C03645=1190.847,-75.511,-40.674,179.388,5.625,149.176
C03646=1190.842,-75.240,-40.686,179.390,5.625,149.175
C03647=1190.836,-74.969,-40.698,179.392,5.625,149.174
C03648=1190.830,-74.720,-40.709,179.395,5.625,149.173
C03649=1190.826,-74.470,-40.720,179.397,5.625,149.173
C03650=1190.820,-74.220,-40.730,179.399,5.626,149.172
C03651=1190.815,-73.970,-40.741,179.402,5.626,149.172
C03652=1190.810,-73.721,-40.752,179.404,5.626,149.171
C03653=1190.804,-73.471,-40.763,179.406,5.627,149.170
C03654=1190.799,-73.222,-40.774,179.409,5.627,149.170
C03655=1190.794,-72.972,-40.784,179.411,5.627,149.169
C03656=1190.789,-72.722,-40.796,179.413,5.627,149.168
C03657=1190.783,-72.472,-40.806,179.415,5.627,149.168
C03658=1190.779,-72.223,-40.817,179.418,5.628,149.167
C03659=1190.772,-71.973,-40.828,179.420,5.628,149.167
C03660=1190.768,-71.723,-40.839,179.422,5.628,149.166
C03661=1190.763,-71.473,-40.850,179.425,5.628,149.165
C03662=1190.757,-71.224,-40.861,179.428,5.629,149.164
C03663=1190.752,-70.974,-40.871,179.429,5.629,149.164
C03664=1190.746,-70.725,-40.883,179.432,5.629,149.163
C03665=1190.741,-70.474,-40.893,179.435,5.630,149.163
C03666=1190.737,-70.225,-40.905,179.436,5.630,149.162
C03667=1190.731,-69.976,-40.915,179.439,5.630,149.161
C03668=1190.726,-69.725,-40.927,179.441,5.630,149.161
C03669=1190.720,-69.476,-40.938,179.444,5.630,149.160
C03670=1190.715,-69.226,-40.948,179.446,5.631,149.159
C03671=1190.711,-68.976,-40.959,179.448,5.631,149.159
C03672=1190.704,-68.727,-40.970,179.451,5.631,149.158
C03673=1190.700,-68.477,-40.982,179.453,5.632,149.158
C03674=1190.695,-68.227,-40.993,179.455,5.631,149.157
C03675=1190.689,-67.978,-41.003,179.457,5.632,149.156
C03676=1190.684,-67.728,-41.015,179.460,5.632,149.155
C03677=1190.679,-67.478,-41.026,179.462,5.632,149.155
C03678=1190.674,-67.229,-41.036,179.464,5.633,149.154
C03679=1190.668,-66.979,-41.048,179.466,5.632,149.154
C03680=1190.663,-66.729,-41.059,179.469,5.633,149.153
C03681=1190.658,-66.480,-41.070,179.471,5.634,149.152
C03682=1190.653,-66.230,-41.081,179.473,5.633,149.152
C03683=1190.648,-65.979,-41.092,179.476,5.634,149.151
C03684=1190.642,-65.731,-41.103,179.478,5.634,149.151
C03685=1190.638,-65.481,-41.114,179.480,5.634,149.150
C03686=1190.632,-65.230,-41.126,179.483,5.635,149.149
C03687=1190.626,-64.981,-41.137,179.486,5.635,149.148
C03688=1190.622,-64.732,-41.148,179.487,5.635,149.148
C03689=1190.616,-64.482,-41.160,179.490,5.635,149.147
C03690=1190.611,-64.232,-41.170,179.493,5.636,149.147
C03691=1190.606,-63.983,-41.181,179.494,5.636,149.146
C03692=1190.601,-63.733,-41.193,179.497,5.636,149.145
C03693=1190.595,-63.484,-41.204,179.500,5.637,149.145
C03694=1190.590,-63.233,-41.215,179.502,5.636,149.144
C03695=1190.585,-62.984,-41.227,179.504,5.637,149.143
C03696=1190.580,-62.734,-41.238,179.506,5.638,149.143
C03697=1190.574,-62.485,-41.249,179.509,5.637,149.142
C03698=1190.569,-62.235,-41.260,179.511,5.638,149.141
C03699=1190.565,-61.985,-41.271,179.513,5.638,149.141
C03700=1190.559,-61.735,-41.283,179.515,5.638,149.140
C03701=1190.554,-61.486,-41.294,179.518,5.638,149.139
C03702=1190.548,-61.236,-41.306,179.520,5.639,149.139
C03703=1190.543,-60.986,-41.316,179.522,5.639,149.138
C03704=1190.539,-60.736,-41.328,179.525,5.639,149.138
C03705=1190.533,-60.487,-41.339,179.528,5.640,149.137
C03706=1190.528,-60.237,-41.351,179.529,5.640,149.136
C03707=1190.523,-59.987,-41.362,179.532,5.640,149.136
C03708=1190.518,-59.738,-41.374,179.535,5.641,149.135
C03709=1190.512,-59.488,-41.385,179.537,5.640,149.134
C03710=1190.507,-59.238,-41.396,179.539,5.641,149.134
C03711=1190.501,-58.988,-41.408,179.542,5.642,149.133
C03712=1190.497,-58.739,-41.419,179.544,5.641,149.132
C03713=1190.491,-58.490,-41.430,179.546,5.642,149.132
C03714=1190.486,-58.240,-41.442,179.549,5.642,149.131
C03715=1190.481,-57.990,-41.453,179.551,5.642,149.130
C03716=1190.476,-57.740,-41.465,179.553,5.642,149.130
C03717=1190.471,-57.491,-41.476,179.556,5.643,149.129
C03718=1190.465,-57.242,-41.488,179.558,5.643,149.129
C03719=1190.460,-56.991,-41.498,179.560,5.643,149.128
C03720=1190.455,-56.741,-41.510,179.563,5.644,149.127
C03721=1190.450,-56.492,-41.522,179.565,5.645,149.127
C03722=1190.445,-56.242,-41.533,179.567,5.644,149.126
C03723=1190.440,-55.992,-41.545,179.570,5.645,149.125
C03724=1190.434,-55.743,-41.556,179.573,5.645,149.125
C03725=1190.429,-55.493,-41.568,179.574,5.645,149.124
C03726=1190.424,-55.243,-41.579,179.577,5.646,149.123
C03727=1190.419,-54.994,-41.591,179.579,5.646,149.123
C03728=1190.414,-54.744,-41.603,179.581,5.646,149.122
C03729=1190.409,-54.494,-41.614,179.584,5.646,149.122
C03730=1190.403,-54.245,-41.625,179.586,5.647,149.121
C03731=1190.397,-53.995,-41.637,179.588,5.647,149.120
C03732=1190.393,-53.745,-41.649,179.591,5.647,149.119
C03733=1190.387,-53.495,-41.660,179.593,5.648,149.119
C03734=1190.383,-53.246,-41.672,179.596,5.648,149.118
C03735=1190.377,-52.996,-41.684,179.598,5.648,149.118
C03736=1190.373,-52.746,-41.695,179.601,5.648,149.117
C03737=1190.367,-52.498,-41.707,179.603,5.649,149.116
C03738=1190.361,-52.248,-41.719,179.605,5.649,149.116
C03739=1190.357,-51.998,-41.730,179.608,5.649,149.115
C03740=1190.351,-51.748,-41.742,179.610,5.650,149.114
C03741=1190.347,-51.498,-41.754,179.612,5.650,149.114
C03742=1190.341,-51.249,-41.765,179.615,5.650,149.113
C03743=1190.336,-50.999,-41.777,179.617,5.651,149.112
C03744=1190.331,-50.749,-41.789,179.620,5.651,149.112
C03745=1190.325,-50.500,-41.800,179.621,5.651,149.111
C03746=1190.320,-50.250,-41.812,179.624,5.651,149.110
C03747=1190.315,-50.001,-41.824,179.627,5.652,149.110
C03748=1190.310,-49.730,-41.836,179.629,5.652,149.109
C03749=1190.304,-49.460,-41.849,179.632,5.652,149.108
C03750=1190.298,-49.190,-41.862,179.634,5.652,149.108
C03751=1190.293,-48.919,-41.875,179.637,5.653,149.107
C03752=1190.288,-48.670,-41.887,179.640,5.653,149.106
C03753=1190.282,-48.420,-41.899,179.642,5.654,149.106
C03754=1190.277,-48.171,-41.909,179.644,5.654,149.105
C03755=1190.272,-47.921,-41.922,179.646,5.654,149.104
C03756=1190.266,-47.671,-41.934,179.649,5.655,149.104
C03757=1190.262,-47.422,-41.945,179.651,5.655,149.103
C03758=1190.256,-47.172,-41.957,179.653,5.655,149.103
C03759=1190.251,-46.922,-41.969,179.656,5.656,149.102
C03760=1190.246,-46.673,-41.982,179.659,5.656,149.101
C03761=1190.241,-46.423,-41.993,179.660,5.656,149.101
C03762=1190.236,-46.173,-42.005,179.663,5.656,149.100
C03763=1190.230,-45.923,-42.017,179.666,5.657,149.099
C03764=1190.225,-45.674,-42.029,179.668,5.657,149.099
C03765=1190.220,-45.424,-42.041,179.670,5.657,149.098
C03766=1190.215,-45.174,-42.052,179.673,5.658,149.097
C03767=1190.210,-44.925,-42.065,179.675,5.658,149.097
C03768=1190.204,-44.675,-42.077,179.677,5.658,149.096
C03769=1190.200,-44.425,-42.088,179.679,5.659,149.095
C03770=1190.194,-44.175,-42.100,179.682,5.659,149.095
C03771=1190.189,-43.926,-42.113,179.685,5.660,149.094
C03772=1190.184,-43.676,-42.125,179.687,5.659,149.093
C03773=1190.179,-43.427,-42.136,179.689,5.660,149.093
C03774=1190.174,-43.177,-42.148,179.692,5.660,149.092
C03775=1190.168,-42.927,-42.160,179.694,5.661,149.091
C03776=1190.163,-42.677,-42.172,179.696,5.661,149.091
C03777=1190.158,-42.428,-42.185,179.699,5.661,149.090
C03778=1190.153,-42.178,-42.196,179.701,5.662,149.090
C03779=1190.148,-41.929,-42.209,179.704,5.662,149.089
C03780=1190.143,-41.679,-42.221,179.706,5.662,149.088
C03781=1190.137,-41.429,-42.233,179.708,5.663,149.088
C03782=1190.132,-41.180,-42.245,179.711,5.663,149.087
C03783=1190.127,-40.930,-42.257,179.714,5.664,149.086
C03784=1190.122,-40.681,-42.269,179.716,5.663,149.086
C03785=1190.117,-40.431,-42.281,179.718,5.664,149.085
C03786=1190.111,-40.181,-42.293,179.721,5.665,149.084
C03787=1190.106,-39.932,-42.305,179.723,5.665,149.084
C03788=1190.101,-39.682,-42.317,179.725,5.665,149.083
C03789=1190.096,-39.433,-42.330,179.728,5.665,149.082
C03790=1190.090,-39.183,-42.342,179.730,5.666,149.082
C03791=1190.086,-38.934,-42.354,179.733,5.666,149.081
C03792=1190.080,-38.684,-42.366,179.735,5.666,149.080
C03793=1190.075,-38.434,-42.378,179.737,5.666,149.080
C03794=1190.070,-38.184,-42.390,179.740,5.667,149.079
C03795=1190.065,-37.935,-42.403,179.742,5.668,149.079
C03796=1190.059,-37.685,-42.415,179.744,5.667,149.078
C03797=1190.055,-37.435,-42.428,179.747,5.668,149.077
C03798=1190.049,-37.185,-42.439,179.749,5.669,149.077
C03799=1190.044,-36.936,-42.452,179.752,5.669,149.076
C03800=1190.039,-36.686,-42.464,179.754,5.669,149.075
C03801=1190.034,-36.437,-42.477,179.757,5.669,149.075
C03802=1190.028,-36.187,-42.488,179.759,5.670,149.074
C03803=1190.024,-35.938,-42.500,179.761,5.670,149.073
C03804=1190.018,-35.688,-42.512,179.764,5.671,149.073
C03805=1190.013,-35.438,-42.525,179.766,5.671,149.072
C03806=1190.008,-35.189,-42.538,179.768,5.671,149.072
C03807=1190.003,-34.938,-42.550,179.771,5.672,149.071
C03808=1189.998,-34.689,-42.562,179.774,5.672,149.070
C03809=1189.993,-34.439,-42.574,179.776,5.672,149.070
C03810=1189.988,-34.190,-42.587,179.778,5.672,149.069
C03811=1189.983,-33.941,-42.599,179.781,5.673,149.068
C03812=1189.977,-33.691,-42.611,179.783,5.674,149.068
C03813=1189.972,-33.441,-42.624,179.786,5.674,149.067
C03814=1189.967,-33.192,-42.637,179.788,5.674,149.066
C03815=1189.962,-32.941,-42.649,179.790,5.675,149.066
C03816=1189.957,-32.692,-42.661,179.793,5.675,149.065
C03817=1189.952,-32.442,-42.673,179.796,5.676,149.064
C03818=1189.946,-32.193,-42.686,179.798,5.675,149.064
C03819=1189.941,-31.943,-42.698,179.800,5.676,149.063
C03820=1189.936,-31.694,-42.711,179.802,5.676,149.063
C03821=1189.931,-31.444,-42.723,179.805,5.677,149.062
C03822=1189.925,-31.194,-42.737,179.808,5.677,149.061
C03823=1189.920,-30.945,-42.749,179.809,5.677,149.061
C03824=1189.915,-30.695,-42.761,179.812,5.678,149.060
C03825=1189.910,-30.445,-42.774,179.815,5.678,149.059
C03826=1189.905,-30.196,-42.786,179.817,5.679,149.059
C03827=1189.900,-29.946,-42.799,179.820,5.680,149.058
C03828=1189.895,-29.696,-42.811,179.822,5.679,149.057
C03829=1189.890,-29.447,-42.824,179.824,5.680,149.057
C03830=1189.884,-29.197,-42.836,179.827,5.680,149.056
C03831=1189.879,-28.948,-42.849,179.830,5.681,149.055
C03832=1189.874,-28.697,-42.861,179.832,5.681,149.055
C03833=1189.869,-28.448,-42.874,179.834,5.681,149.054
C03834=1189.864,-28.198,-42.887,179.837,5.682,149.053
C03835=1189.858,-27.949,-42.900,179.839,5.682,149.053
C03836=1189.853,-27.700,-42.912,179.841,5.683,149.052
C03837=1189.848,-27.449,-42.924,179.844,5.683,149.052
C03838=1189.843,-27.200,-42.937,179.846,5.683,149.051
C03839=1189.838,-26.951,-42.950,179.849,5.683,149.050
C03840=1189.833,-26.701,-42.962,179.851,5.684,149.050
C03841=1189.829,-26.451,-42.975,179.854,5.685,149.049
C03842=1189.823,-26.202,-42.988,179.856,5.685,149.048
C03843=1189.817,-25.952,-43.000,179.858,5.685,149.048
C03844=1189.812,-25.702,-43.013,179.860,5.686,149.047
C03845=1189.808,-25.452,-43.026,179.863,5.686,149.046
C03846=1189.802,-25.203,-43.038,179.866,5.687,149.046
C03847=1189.797,-24.954,-43.051,179.868,5.687,149.045
C03848=1189.791,-24.704,-43.064,179.871,5.688,149.044
C03849=1189.787,-24.454,-43.077,179.873,5.688,149.044
C03850=1189.782,-24.205,-43.090,179.875,5.688,149.043
C03851=1189.777,-23.955,-43.102,179.878,5.688,149.042
C03852=1189.771,-23.685,-43.117,179.881,5.689,149.042
C03853=1189.766,-23.416,-43.130,179.883,5.689,149.041
C03854=1189.760,-23.146,-43.144,179.886,5.690,149.040
C03855=1189.755,-22.877,-43.158,179.889,5.690,149.040
C03856=1189.750,-22.627,-43.171,179.891,5.691,149.039
C03857=1189.744,-22.378,-43.184,179.894,5.692,149.039
C03858=1189.739,-22.128,-43.197,179.896,5.691,149.038
C03859=1189.734,-21.878,-43.209,179.898,5.692,149.037
C03860=1189.729,-21.629,-43.222,179.901,5.692,149.036
C03861=1189.724,-21.379,-43.235,179.903,5.693,149.036
C03862=1189.718,-21.129,-43.248,179.906,5.693,149.035
C03863=1189.713,-20.880,-43.261,179.908,5.694,149.035
C03864=1189.709,-20.630,-43.274,179.910,5.694,149.034
C03865=1189.703,-20.380,-43.287,179.913,5.694,149.033
C03866=1189.698,-20.131,-43.299,179.915,5.695,149.033
C03867=1189.693,-19.881,-43.312,179.918,5.695,149.032
C03868=1189.687,-19.631,-43.326,179.921,5.696,149.031
C03869=1189.682,-19.382,-43.338,179.923,5.696,149.031
C03870=1189.678,-19.132,-43.351,179.925,5.696,149.030
C03871=1189.672,-18.882,-43.364,179.928,5.697,149.030
C03872=1189.667,-18.633,-43.377,179.930,5.697,149.029
C03873=1189.662,-18.383,-43.390,179.933,5.698,149.028
C03874=1189.656,-18.133,-43.403,179.935,5.699,149.028
C03875=1189.651,-17.884,-43.416,179.938,5.699,149.027
C03876=1189.647,-17.635,-43.429,179.940,5.700,149.026
C03877=1189.641,-17.385,-43.443,179.942,5.699,149.026
C03878=1189.636,-17.136,-43.455,179.945,5.700,149.025
C03879=1189.632,-16.886,-43.468,179.947,5.700,149.024
C03880=1189.626,-16.636,-43.481,179.950,5.701,149.024
C03881=1189.621,-16.386,-43.494,179.953,5.701,149.023
C03882=1189.615,-16.137,-43.507,179.955,5.702,149.023
C03883=1189.611,-15.888,-43.521,179.957,5.703,149.022
C03884=1189.606,-15.638,-43.534,179.959,5.702,149.021
C03885=1189.600,-15.388,-43.547,179.962,5.703,149.020
C03886=1189.596,-15.138,-43.560,179.965,5.703,149.020
C03887=1189.590,-14.889,-43.573,179.967,5.704,149.019
C03888=1189.585,-14.640,-43.586,179.970,5.705,149.019
C03889=1189.580,-14.390,-43.599,179.972,5.705,149.018
C03890=1189.575,-14.140,-43.613,179.975,5.706,149.017
C03891=1189.570,-13.890,-43.626,179.977,5.706,149.017
C03892=1189.564,-13.641,-43.639,179.979,5.706,149.016
C03893=1189.560,-13.391,-43.652,179.982,5.707,149.015
C03894=1189.554,-13.142,-43.666,179.984,5.707,149.015
C03895=1189.549,-12.892,-43.678,179.987,5.708,149.014
C03896=1189.545,-12.643,-43.692,179.989,5.708,149.014
C03897=1189.539,-12.393,-43.705,179.992,5.709,149.013
C03898=1189.534,-12.143,-43.718,179.995,5.709,149.012
C03899=1189.529,-11.894,-43.732,179.996,5.709,149.012
C03900=1189.524,-11.644,-43.745,179.999,5.710,149.011
C03901=1189.518,-11.394,-43.758,-179.998,5.710,149.010
C03902=1189.514,-11.145,-43.772,-179.996,5.711,149.010
C03903=1189.508,-10.895,-43.785,-179.994,5.712,149.009
C03904=1189.504,-10.645,-43.798,-179.991,5.712,149.008
C03905=1189.498,-10.396,-43.812,-179.988,5.712,149.008
C03906=1189.494,-10.146,-43.825,-179.986,5.713,149.007
C03907=1189.488,-9.897,-43.838,-179.984,5.713,149.006
C03908=1189.484,-9.647,-43.852,-179.981,5.713,149.006
C03909=1189.478,-9.398,-43.865,-179.979,5.714,149.005
C03910=1189.473,-9.148,-43.878,-179.976,5.714,149.005
C03911=1189.468,-8.899,-43.892,-179.973,5.715,149.004
C03912=1189.463,-8.649,-43.905,-179.971,5.716,149.003
C03913=1189.458,-8.400,-43.919,-179.969,5.716,149.003
C03914=1189.452,-8.149,-43.932,-179.966,5.717,149.002
C03915=1189.448,-7.901,-43.946,-179.963,5.717,149.001
C03916=1189.442,-7.650,-43.959,-179.962,5.717,149.001
C03917=1189.437,-7.401,-43.972,-179.959,5.718,149.000
C03918=1189.432,-7.151,-43.986,-179.956,5.718,148.999
C03919=1189.427,-6.902,-43.999,-179.954,5.719,148.999
C03920=1189.422,-6.652,-44.013,-179.952,5.719,148.998
C03921=1189.416,-6.403,-44.026,-179.949,5.720,148.998
C03922=1189.412,-6.153,-44.040,-179.946,5.720,148.997
C03923=1189.406,-5.904,-44.053,-179.944,5.721,148.996
C03924=1189.402,-5.654,-44.067,-179.941,5.722,148.996
C03925=1189.396,-5.405,-44.080,-179.939,5.722,148.995
C03926=1189.391,-5.155,-44.094,-179.936,5.723,148.994
C03927=1189.387,-4.905,-44.107,-179.934,5.722,148.994
C03928=1189.381,-4.656,-44.121,-179.932,5.723,148.993
C03929=1189.376,-4.406,-44.135,-179.929,5.724,148.993
C03930=1189.371,-4.157,-44.148,-179.927,5.724,148.992
C03931=1189.366,-3.907,-44.162,-179.924,5.725,148.991
C03932=1189.360,-3.657,-44.175,-179.922,5.725,148.991
C03933=1189.356,-3.408,-44.189,-179.919,5.726,148.990
C03934=1189.351,-3.158,-44.203,-179.916,5.726,148.989
C03935=1189.345,-2.909,-44.217,-179.914,5.727,148.989
C03936=1189.341,-2.659,-44.230,-179.911,5.727,148.988
C03937=1189.335,-2.410,-44.243,-179.909,5.728,148.987
C03938=1189.330,-2.160,-44.258,-179.906,5.729,148.987
C03939=1189.326,-1.910,-44.271,-179.904,5.728,148.986
C03940=1189.320,-1.661,-44.285,-179.902,5.729,148.985
C03941=1189.315,-1.411,-44.299,-179.899,5.730,148.985
C03942=1189.309,-1.162,-44.312,-179.897,5.730,148.984
C03943=1189.305,-0.912,-44.326,-179.894,5.731,148.984
C03944=1189.300,-0.663,-44.340,-179.891,5.731,148.983
C03945=1189.294,-0.413,-44.353,-179.889,5.732,148.982
C03946=1189.289,-0.163,-44.367,-179.887,5.733,148.982
C03947=1189.285,0.086,-44.381,-179.884,5.733,148.981
C03948=1189.279,0.336,-44.394,-179.881,5.733,148.980
C03949=1189.274,0.586,-44.409,-179.879,5.734,148.980
C03950=1189.269,0.835,-44.423,-179.877,5.735,148.979
C03951=1189.264,1.085,-44.436,-179.874,5.735,148.979
C03952=1189.259,1.334,-44.450,-179.871,5.736,148.978
C03953=1189.254,1.583,-44.464,-179.869,5.737,148.977
C03954=1189.249,1.833,-44.478,-179.867,5.736,148.977
C03955=1189.243,2.083,-44.492,-179.864,5.737,148.976
C03956=1189.238,2.351,-44.506,-179.861,5.738,148.975
C03957=1189.233,2.621,-44.521,-179.858,5.739,148.975
C03958=1189.228,2.890,-44.536,-179.856,5.739,148.974
C03959=1189.222,3.159,-44.551,-179.853,5.739,148.973
C03960=1189.217,3.409,-44.566,-179.851,5.740,148.973
C03961=1189.212,3.658,-44.579,-179.848,5.741,148.972
C03962=1189.206,3.908,-44.593,-179.846,5.741,148.971
C03963=1189.201,4.158,-44.607,-179.843,5.742,148.971
C03964=1189.197,4.407,-44.621,-179.841,5.743,148.970
C03965=1189.192,4.657,-44.635,-179.838,5.743,148.970
C03966=1189.187,4.906,-44.649,-179.836,5.743,148.969
C03967=1189.181,5.155,-44.663,-179.833,5.743,148.968
C03968=1189.176,5.406,-44.677,-179.831,5.744,148.968
C03969=1189.171,5.655,-44.691,-179.829,5.745,148.967
C03970=1189.166,5.905,-44.705,-179.826,5.745,148.966
C03971=1189.160,6.154,-44.719,-179.823,5.746,148.966
C03972=1189.156,6.403,-44.733,-179.821,5.746,148.965
C03973=1189.151,6.653,-44.747,-179.819,5.747,148.965
C03974=1189.146,6.903,-44.761,-179.816,5.747,148.964
C03975=1189.141,7.152,-44.775,-179.813,5.748,148.963
C03976=1189.136,7.402,-44.790,-179.811,5.749,148.963
C03977=1189.131,7.651,-44.804,-179.808,5.749,148.962
C03978=1189.126,7.901,-44.818,-179.806,5.750,148.961
C03979=1189.120,8.150,-44.832,-179.803,5.750,148.961
C03980=1189.115,8.400,-44.846,-179.801,5.751,148.960
C03981=1189.110,8.650,-44.860,-179.798,5.752,148.960
C03982=1189.105,8.900,-44.874,-179.796,5.752,148.959
C03983=1189.100,9.149,-44.888,-179.793,5.753,148.958
C03984=1189.095,9.398,-44.902,-179.791,5.753,148.958
C03985=1189.090,9.648,-44.917,-179.788,5.754,148.957
C03986=1189.085,9.898,-44.931,-179.786,5.754,148.956
C03987=1189.080,10.148,-44.945,-179.783,5.755,148.956
C03988=1189.074,10.397,-44.959,-179.781,5.756,148.955
C03989=1189.070,10.646,-44.974,-179.778,5.756,148.954
C03990=1189.065,10.895,-44.988,-179.775,5.757,148.954
C03991=1189.060,11.145,-45.003,-179.773,5.758,148.953
C03992=1189.055,11.395,-45.017,-179.771,5.758,148.953
C03993=1189.049,11.644,-45.031,-179.768,5.759,148.952
C03994=1189.044,11.894,-45.045,-179.765,5.759,148.951
C03995=1189.039,12.143,-45.059,-179.763,5.760,148.951
C03996=1189.034,12.393,-45.074,-179.760,5.760,148.950
C03997=1189.029,12.643,-45.088,-179.758,5.761,148.949
C03998=1189.024,12.892,-45.102,-179.755,5.761,148.949
C03999=1189.019,13.141,-45.116,-179.753,5.762,148.948
C04000=1189.014,13.391,-45.130,-179.750,5.763,148.948
C04001=1189.009,13.640,-45.145,-179.748,5.763,148.947
C04002=1189.004,13.890,-45.160,-179.745,5.764,148.946
C04003=1188.999,14.140,-45.174,-179.743,5.765,148.946
C04004=1188.994,14.389,-45.188,-179.740,5.765,148.945
C04005=1188.989,14.638,-45.202,-179.738,5.766,148.944
C04006=1188.984,14.888,-45.216,-179.735,5.766,148.944
C04007=1188.978,15.137,-45.232,-179.733,5.767,148.943
C04008=1188.973,15.387,-45.246,-179.730,5.767,148.943
C04009=1188.969,15.637,-45.260,-179.727,5.768,148.942
C04010=1188.964,15.887,-45.275,-179.725,5.769,148.941
C04011=1188.959,16.136,-45.289,-179.723,5.769,148.941
C04012=1188.954,16.385,-45.304,-179.720,5.770,148.940
C04013=1188.948,16.634,-45.318,-179.717,5.770,148.939
C04014=1188.943,16.884,-45.332,-179.715,5.771,148.939
C04015=1188.938,17.134,-45.347,-179.713,5.772,148.938
C04016=1188.933,17.383,-45.362,-179.710,5.772,148.938
C04017=1188.928,17.633,-45.376,-179.708,5.773,148.937
C04018=1188.923,17.883,-45.391,-179.705,5.773,148.936
C04019=1188.918,18.132,-45.405,-179.702,5.774,148.936
C04020=1188.914,18.381,-45.420,-179.700,5.774,148.935
C04021=1188.908,18.631,-45.435,-179.698,5.775,148.935
C04022=1188.903,18.881,-45.449,-179.695,5.776,148.934
C04023=1188.898,19.130,-45.464,-179.692,5.776,148.933
C04024=1188.893,19.379,-45.478,-179.690,5.777,148.933
C04025=1188.888,19.629,-45.492,-179.688,5.778,148.932
C04026=1188.882,19.878,-45.508,-179.685,5.778,148.931
C04027=1188.877,20.128,-45.522,-179.682,5.779,148.931
C04028=1188.873,20.378,-45.536,-179.680,5.780,148.930
C04029=1188.868,20.627,-45.551,-179.677,5.780,148.930
C04030=1188.863,20.877,-45.566,-179.675,5.780,148.929
C04031=1188.858,21.126,-45.581,-179.672,5.781,148.928
C04032=1188.853,21.376,-45.596,-179.669,5.783,148.928
C04033=1188.848,21.625,-45.610,-179.667,5.783,148.927
C04034=1188.843,21.874,-45.625,-179.664,5.784,148.926
C04035=1188.837,22.125,-45.640,-179.662,5.785,148.926
C04036=1188.833,22.374,-45.655,-179.659,5.785,148.925
C04037=1188.828,22.623,-45.669,-179.657,5.786,148.925
C04038=1188.822,22.873,-45.685,-179.654,5.786,148.924
C04039=1188.817,23.122,-45.699,-179.652,5.787,148.924
C04040=1188.812,23.372,-45.713,-179.649,5.787,148.923
C04041=1188.808,23.621,-45.728,-179.647,5.788,148.922
C04042=1188.802,23.871,-45.743,-179.644,5.789,148.922
C04043=1188.797,24.120,-45.758,-179.642,5.789,148.921
C04044=1188.792,24.370,-45.772,-179.639,5.790,148.920
C04045=1188.787,24.619,-45.788,-179.636,5.790,148.920
C04046=1188.782,24.869,-45.802,-179.634,5.791,148.919
C04047=1188.777,25.118,-45.817,-179.632,5.792,148.919
C04048=1188.772,25.368,-45.833,-179.629,5.792,148.918
C04049=1188.767,25.617,-45.847,-179.627,5.793,148.917
C04050=1188.762,25.866,-45.862,-179.624,5.794,148.917
C04051=1188.757,26.116,-45.877,-179.621,5.795,148.916
C04052=1188.752,26.366,-45.892,-179.618,5.795,148.915
C04053=1188.747,26.615,-45.906,-179.616,5.796,148.915
C04054=1188.742,26.865,-45.922,-179.613,5.797,148.914
C04055=1188.737,27.114,-45.936,-179.611,5.797,148.914
C04056=1188.731,27.364,-45.952,-179.609,5.798,148.913
C04057=1188.727,27.613,-45.967,-179.606,5.799,148.912
C04058=1188.722,27.863,-45.981,-179.603,5.799,148.912
C04059=1188.717,28.113,-45.997,-179.601,5.800,148.911
C04060=1188.712,28.382,-46.012,-179.599,5.800,148.911
C04061=1188.706,28.651,-46.029,-179.595,5.802,148.910
C04062=1188.701,28.919,-46.045,-179.593,5.802,148.909
C04063=1188.695,29.188,-46.061,-179.590,5.803,148.909
C04064=1188.691,29.437,-46.076,-179.587,5.803,148.908
C04065=1188.685,29.687,-46.091,-179.585,5.804,148.907
C04066=1188.680,29.936,-46.106,-179.583,5.805,148.907
C04067=1188.675,30.185,-46.122,-179.580,5.805,148.906
C04068=1188.670,30.435,-46.136,-179.577,5.806,148.905
C04069=1188.665,30.685,-46.152,-179.575,5.807,148.905
C04070=1188.660,30.934,-46.167,-179.572,5.808,148.904
C04071=1188.655,31.183,-46.182,-179.569,5.808,148.904
C04072=1188.650,31.434,-46.197,-179.567,5.809,148.903
C04073=1188.645,31.683,-46.213,-179.564,5.810,148.903
C04074=1188.640,31.932,-46.228,-179.562,5.810,148.902
C04075=1188.635,32.181,-46.243,-179.560,5.811,148.901
C04076=1188.630,32.431,-46.257,-179.557,5.812,148.901
C04077=1188.624,32.681,-46.273,-179.554,5.812,148.900
C04078=1188.620,32.930,-46.288,-179.551,5.813,148.899
C04079=1188.615,33.180,-46.304,-179.549,5.814,148.899
C04080=1188.610,33.429,-46.319,-179.546,5.815,148.898
C04081=1188.605,33.679,-46.334,-179.544,5.815,148.898
C04082=1188.600,33.928,-46.349,-179.542,5.816,148.897
C04083=1188.595,34.177,-46.364,-179.539,5.817,148.896
C04084=1188.590,34.426,-46.379,-179.536,5.817,148.896
C04085=1188.585,34.677,-46.395,-179.534,5.818,148.895
C04086=1188.580,34.926,-46.411,-179.531,5.819,148.895
C04087=1188.575,35.176,-46.425,-179.528,5.820,148.894
C04088=1188.569,35.425,-46.441,-179.526,5.821,148.894
C04089=1188.565,35.674,-46.456,-179.523,5.821,148.893
C04090=1188.559,35.924,-46.471,-179.521,5.822,148.892
C04091=1188.555,36.173,-46.487,-179.519,5.823,148.892
C04092=1188.550,36.423,-46.502,-179.516,5.823,148.891
C04093=1188.545,36.672,-46.518,-179.513,5.824,148.890
C04094=1188.540,36.921,-46.533,-179.511,5.824,148.890
C04095=1188.535,37.171,-46.549,-179.508,5.826,148.889
C04096=1188.530,37.421,-46.564,-179.505,5.826,148.889
C04097=1188.525,37.670,-46.579,-179.503,5.827,148.888
C04098=1188.520,37.919,-46.595,-179.501,5.828,148.887
C04099=1188.514,38.169,-46.611,-179.498,5.828,148.887
C04100=1188.510,38.418,-46.626,-179.495,5.829,148.886
C04101=1188.505,38.668,-46.642,-179.493,5.830,148.886
C04102=1188.500,38.917,-46.657,-179.490,5.830,148.885
C04103=1188.495,39.166,-46.672,-179.487,5.832,148.884
C04104=1188.490,39.416,-46.688,-179.485,5.832,148.884
C04105=1188.485,39.666,-46.704,-179.482,5.833,148.883
C04106=1188.480,39.915,-46.719,-179.480,5.833,148.883
C04107=1188.475,40.164,-46.734,-179.478,5.834,148.882
C04108=1188.470,40.414,-46.750,-179.475,5.835,148.881
C04109=1188.465,40.664,-46.766,-179.472,5.835,148.881
C04110=1188.460,40.913,-46.781,-179.470,5.837,148.880
C04111=1188.455,41.162,-46.796,-179.467,5.838,148.880
C04112=1188.450,41.412,-46.812,-179.464,5.838,148.879
C04113=1188.445,41.661,-46.827,-179.462,5.839,148.879
C04114=1188.440,41.911,-46.843,-179.460,5.839,148.878
C04115=1188.435,42.161,-46.859,-179.457,5.840,148.877
C04116=1188.430,42.410,-46.875,-179.454,5.842,148.877
C04117=1188.425,42.659,-46.890,-179.452,5.842,148.876
C04118=1188.420,42.908,-46.906,-179.449,5.843,148.875
C04119=1188.415,43.158,-46.922,-179.447,5.844,148.875
C04120=1188.410,43.408,-46.937,-179.444,5.844,148.874
C04121=1188.404,43.657,-46.953,-179.441,5.845,148.874
C04122=1188.400,43.907,-46.968,-179.439,5.846,148.873
C04123=1188.395,44.156,-46.985,-179.436,5.847,148.872
C04124=1188.390,44.405,-47.000,-179.433,5.847,148.872
C04125=1188.385,44.655,-47.016,-179.431,5.848,148.871
C04126=1188.380,44.905,-47.032,-179.429,5.849,148.871
C04127=1188.375,45.154,-47.047,-179.426,5.849,148.870
C04128=1188.370,45.403,-47.063,-179.423,5.851,148.870
C04129=1188.365,45.653,-47.079,-179.421,5.851,148.869
C04130=1188.360,45.902,-47.095,-179.418,5.852,148.868
C04131=1188.355,46.152,-47.111,-179.416,5.853,148.868
C04132=1188.350,46.401,-47.127,-179.413,5.853,148.867
C04133=1188.345,46.651,-47.143,-179.411,5.854,148.866
C04134=1188.340,46.900,-47.158,-179.408,5.856,148.866
C04135=1188.335,47.149,-47.174,-179.405,5.856,148.865
C04136=1188.330,47.399,-47.190,-179.403,5.857,148.865
C04137=1188.325,47.648,-47.206,-179.400,5.857,148.864
C04138=1188.320,47.898,-47.221,-179.398,5.858,148.864
C04139=1188.315,48.147,-47.238,-179.395,5.860,148.863
C04140=1188.310,48.397,-47.253,-179.392,5.860,148.862
C04141=1188.305,48.647,-47.269,-179.390,5.861,148.862
C04142=1188.300,48.896,-47.286,-179.388,5.862,148.861
C04143=1188.296,49.145,-47.301,-179.385,5.862,148.861
C04144=1188.291,49.394,-47.317,-179.382,5.863,148.860
C04145=1188.285,49.644,-47.333,-179.380,5.864,148.860
C04146=1188.281,49.894,-47.349,-179.377,5.865,148.859
C04147=1188.276,50.142,-47.365,-179.374,5.865,148.858
C04148=1188.271,50.393,-47.381,-179.372,5.866,148.858
C04149=1188.266,50.641,-47.397,-179.370,5.867,148.857
C04150=1188.261,50.891,-47.413,-179.366,5.868,148.856
C04151=1188.256,51.141,-47.429,-179.364,5.869,148.856
C04152=1188.250,51.390,-47.445,-179.362,5.870,148.855
C04153=1188.246,51.640,-47.461,-179.359,5.870,148.855
C04154=1188.241,51.889,-47.478,-179.356,5.872,148.854
C04155=1188.236,52.139,-47.494,-179.354,5.872,148.854
C04156=1188.231,52.387,-47.510,-179.351,5.873,148.853
C04157=1188.226,52.638,-47.526,-179.349,5.874,148.852
C04158=1188.221,52.886,-47.542,-179.346,5.874,148.852
C04159=1188.216,53.136,-47.558,-179.343,5.876,148.851
C04160=1188.211,53.385,-47.574,-179.341,5.876,148.851
C04161=1188.206,53.635,-47.590,-179.338,5.877,148.850
C04162=1188.201,53.884,-47.607,-179.336,5.878,148.850
C04163=1188.196,54.134,-47.623,-179.333,5.878,148.849
C04164=1188.191,54.402,-47.640,-179.330,5.880,148.848
C04165=1188.186,54.671,-47.657,-179.328,5.881,148.848
C04166=1188.180,54.940,-47.675,-179.325,5.882,148.847
C04167=1188.175,55.208,-47.693,-179.322,5.882,148.846
C04168=1188.169,55.457,-47.709,-179.319,5.883,148.846
C04169=1188.165,55.707,-47.725,-179.317,5.885,148.845
C04170=1188.160,55.956,-47.742,-179.314,5.885,148.845
C04171=1188.155,56.206,-47.758,-179.311,5.886,148.844
C04172=1188.150,56.454,-47.774,-179.309,5.887,148.844
C04173=1188.145,56.705,-47.790,-179.307,5.887,148.843
C04174=1188.140,56.954,-47.806,-179.304,5.889,148.843
C04175=1188.135,57.203,-47.823,-179.301,5.889,148.842
C04176=1188.130,57.453,-47.839,-179.299,5.890,148.841
C04177=1188.125,57.702,-47.856,-179.297,5.891,148.841
C04178=1188.120,57.951,-47.872,-179.293,5.892,148.840
C04179=1188.115,58.201,-47.888,-179.291,5.893,148.839
C04180=1188.110,58.450,-47.905,-179.289,5.894,148.839
C04181=1188.105,58.699,-47.921,-179.286,5.894,148.838
C04182=1188.100,58.949,-47.938,-179.283,5.896,148.838
C04183=1188.095,59.199,-47.954,-179.281,5.896,148.837
C04184=1188.090,59.448,-47.970,-179.278,5.897,148.837
C04185=1188.086,59.697,-47.987,-179.276,5.898,148.836
C04186=1188.080,59.947,-48.003,-179.273,5.899,148.835
C04187=1188.075,60.197,-48.020,-179.270,5.900,148.835
C04188=1188.070,60.445,-48.036,-179.268,5.900,148.834
C04189=1188.066,60.695,-48.053,-179.265,5.901,148.834
C04190=1188.061,60.944,-48.070,-179.262,5.903,148.833
C04191=1188.056,61.194,-48.085,-179.260,5.903,148.833
C04192=1188.051,61.443,-48.102,-179.258,5.904,148.832
C04193=1188.045,61.692,-48.119,-179.254,5.905,148.831
C04194=1188.041,61.942,-48.135,-179.252,5.906,148.831
C04195=1188.037,62.191,-48.152,-179.250,5.907,148.830
C04196=1188.030,62.441,-48.168,-179.247,5.907,148.830
C04197=1188.026,62.690,-48.185,-179.244,5.909,148.829
C04198=1188.021,62.940,-48.202,-179.242,5.910,148.829
C04199=1188.016,63.189,-48.218,-179.239,5.910,148.828
C04200=1188.011,63.438,-48.235,-179.237,5.911,148.828
C04201=1188.007,63.688,-48.252,-179.234,5.912,148.827
C04202=1188.002,63.937,-48.268,-179.231,5.913,148.826
C04203=1187.996,64.187,-48.285,-179.229,5.914,148.826
C04204=1187.992,64.436,-48.302,-179.226,5.915,148.825
C04205=1187.987,64.685,-48.318,-179.223,5.916,148.825
C04206=1187.981,64.935,-48.335,-179.221,5.917,148.824
C04207=1187.977,65.185,-48.352,-179.219,5.918,148.824
C04208=1187.972,65.433,-48.368,-179.215,5.919,148.823
C04209=1187.967,65.683,-48.385,-179.213,5.919,148.822
C04210=1187.962,65.933,-48.402,-179.211,5.920,148.822
C04211=1187.957,66.182,-48.418,-179.208,5.922,148.821
C04212=1187.952,66.431,-48.435,-179.205,5.923,148.821
C04213=1187.947,66.681,-48.452,-179.203,5.923,148.820
C04214=1187.942,66.930,-48.468,-179.201,5.924,148.820
C04215=1187.937,67.179,-48.486,-179.197,5.925,148.819
C04216=1187.932,67.429,-48.502,-179.195,5.926,148.818
C04217=1187.927,67.679,-48.520,-179.193,5.927,148.818
C04218=1187.922,67.927,-48.536,-179.189,5.928,148.817
C04219=1187.918,68.177,-48.552,-179.187,5.929,148.817
C04220=1187.913,68.426,-48.570,-179.185,5.930,148.816
C04221=1187.908,68.675,-48.587,-179.182,5.931,148.816
C04222=1187.902,68.925,-48.604,-179.179,5.932,148.815
C04223=1187.898,69.174,-48.621,-179.177,5.932,148.814
C04224=1187.894,69.424,-48.637,-179.174,5.934,148.814
C04225=1187.888,69.673,-48.654,-179.171,5.935,148.813
C04226=1187.883,69.922,-48.671,-179.169,5.935,148.813
C04227=1187.878,70.172,-48.688,-179.167,5.936,148.812
C04228=1187.874,70.422,-48.705,-179.164,5.938,148.812
C04229=1187.868,70.670,-48.722,-179.161,5.938,148.811
C04230=1187.864,70.919,-48.739,-179.159,5.939,148.810
C04231=1187.858,71.169,-48.756,-179.156,5.941,148.810
C04232=1187.854,71.419,-48.773,-179.153,5.941,148.809
C04233=1187.849,71.669,-48.790,-179.151,5.942,148.809
C04234=1187.844,71.917,-48.807,-179.148,5.943,148.808
C04235=1187.839,72.167,-48.825,-179.146,5.944,148.808
C04236=1187.834,72.416,-48.841,-179.143,5.945,148.807
C04237=1187.829,72.666,-48.859,-179.140,5.946,148.807
C04238=1187.824,72.915,-48.875,-179.138,5.947,148.806
C04239=1187.819,73.164,-48.892,-179.135,5.948,148.805
C04240=1187.814,73.413,-48.910,-179.132,5.949,148.805
C04241=1187.809,73.663,-48.927,-179.130,5.950,148.804
C04242=1187.805,73.913,-48.943,-179.128,5.951,148.804
C04243=1187.800,74.162,-48.961,-179.124,5.952,148.803
C04244=1187.794,74.411,-48.978,-179.122,5.953,148.803
C04245=1187.790,74.660,-48.995,-179.120,5.954,148.802
C04246=1187.784,74.910,-49.012,-179.116,5.955,148.802
C04247=1187.780,75.159,-49.030,-179.114,5.956,148.801
C04248=1187.775,75.409,-49.047,-179.111,5.957,148.800
C04249=1187.770,75.659,-49.064,-179.109,5.958,148.800
C04250=1187.766,75.907,-49.082,-179.106,5.959,148.799
C04251=1187.760,76.156,-49.098,-179.104,5.960,148.799
C04252=1187.755,76.406,-49.115,-179.101,5.961,148.798
C04253=1187.750,76.655,-49.133,-179.099,5.962,148.798
C04254=1187.745,76.905,-49.150,-179.096,5.963,148.797
C04255=1187.741,77.154,-49.168,-179.093,5.964,148.797
C04256=1187.736,77.404,-49.185,-179.091,5.965,148.796
C04257=1187.730,77.653,-49.202,-179.088,5.966,148.795
C04258=1187.726,77.902,-49.220,-179.085,5.967,148.795
C04259=1187.721,78.151,-49.237,-179.083,5.967,148.794
C04260=1187.716,78.401,-49.255,-179.080,5.969,148.794
C04261=1187.711,78.650,-49.271,-179.077,5.970,148.793
C04262=1187.706,78.899,-49.289,-179.075,5.971,148.793
C04263=1187.701,79.149,-49.306,-179.072,5.972,148.792
C04264=1187.697,79.398,-49.324,-179.070,5.973,148.792
C04265=1187.692,79.648,-49.341,-179.067,5.974,148.791
C04266=1187.686,79.897,-49.358,-179.065,5.975,148.791
C04267=1187.682,80.146,-49.376,-179.062,5.976,148.790
C04268=1187.676,80.414,-49.394,-179.059,5.977,148.789
C04269=1187.671,80.683,-49.414,-179.056,5.979,148.789
C04270=1187.666,80.952,-49.432,-179.053,5.979,148.788
C04271=1187.661,81.220,-49.452,-179.050,5.981,148.788
C04272=1187.656,81.469,-49.468,-179.048,5.981,148.787
C04273=1187.651,81.718,-49.486,-179.045,5.982,148.787
C04274=1187.646,81.968,-49.504,-179.043,5.984,148.786
C04275=1187.641,82.217,-49.522,-179.040,5.984,148.786
C04276=1187.635,82.467,-49.538,-179.037,5.986,148.785
C04277=1187.631,82.715,-49.556,-179.035,5.987,148.784
C04278=1187.626,82.965,-49.574,-179.033,5.987,148.784
C04279=1187.621,83.214,-49.591,-179.029,5.989,148.783
C04280=1187.616,83.464,-49.609,-179.027,5.990,148.783
C04281=1187.612,83.712,-49.626,-179.024,5.991,148.782
C04282=1187.607,83.962,-49.644,-179.022,5.992,148.782
C04283=1187.602,84.211,-49.662,-179.019,5.993,148.781
C04284=1187.597,84.461,-49.680,-179.017,5.994,148.781
C04285=1187.592,84.710,-49.697,-179.014,5.995,148.780
C04286=1187.587,84.960,-49.715,-179.011,5.997,148.780
C04287=1187.583,85.208,-49.732,-179.009,5.997,148.779
C04288=1187.577,85.458,-49.750,-179.007,5.998,148.779
C04289=1187.572,85.707,-49.767,-179.003,5.999,148.778
C04290=1187.568,85.957,-49.785,-179.001,6.000,148.778
C04291=1187.562,86.206,-49.803,-178.998,6.002,148.777
C04292=1187.557,86.456,-49.821,-178.996,6.003,148.777
C04293=1187.553,86.705,-49.839,-178.993,6.004,148.776
C04294=1187.548,86.955,-49.857,-178.991,6.005,148.775
C04295=1187.543,87.204,-49.874,-178.988,6.005,148.775
C04296=1187.539,87.453,-49.892,-178.985,6.007,148.774
C04297=1187.534,87.702,-49.910,-178.983,6.008,148.774
C04298=1187.529,87.952,-49.928,-178.980,6.009,148.773
C04299=1187.524,88.201,-49.946,-178.977,6.010,148.773
C04300=1187.519,88.451,-49.963,-178.975,6.011,148.772
C04301=1187.514,88.700,-49.981,-178.972,6.012,148.772
C04302=1187.509,88.949,-49.999,-178.970,6.013,148.771
C04303=1187.504,89.198,-50.017,-178.967,6.014,148.771
C04304=1187.499,89.447,-50.035,-178.964,6.015,148.770
C04305=1187.494,89.696,-50.053,-178.961,6.017,148.769
C04306=1187.489,89.946,-50.071,-178.959,6.018,148.769
C04307=1187.484,90.195,-50.088,-178.956,6.019,148.768
C04308=1187.480,90.445,-50.106,-178.954,6.020,148.768
C04309=1187.475,90.694,-50.124,-178.951,6.020,148.767
C04310=1187.470,90.944,-50.142,-178.948,6.022,148.767
C04311=1187.465,91.193,-50.160,-178.946,6.023,148.766
C04312=1187.460,91.442,-50.178,-178.943,6.024,148.766
C04313=1187.455,91.691,-50.196,-178.940,6.025,148.765
C04314=1187.450,91.940,-50.214,-178.938,6.027,148.765
C04315=1187.445,92.190,-50.232,-178.935,6.027,148.764
C04316=1187.441,92.439,-50.251,-178.932,6.029,148.764
C04317=1187.436,92.689,-50.269,-178.930,6.030,148.763
C04318=1187.431,92.938,-50.287,-178.928,6.031,148.763
C04319=1187.426,93.187,-50.305,-178.925,6.032,148.762
C04320=1187.421,93.436,-50.323,-178.922,6.033,148.762
C04321=1187.417,93.685,-50.340,-178.920,6.035,148.761
C04322=1187.412,93.934,-50.358,-178.917,6.035,148.761
C04323=1187.407,94.184,-50.377,-178.914,6.037,148.760
C04324=1187.402,94.434,-50.395,-178.912,6.037,148.759
C04325=1187.397,94.683,-50.413,-178.909,6.039,148.759
C04326=1187.392,94.932,-50.431,-178.906,6.040,148.758
C04327=1187.387,95.181,-50.449,-178.904,6.041,148.758
C04328=1187.383,95.431,-50.468,-178.901,6.042,148.757
C04329=1187.378,95.680,-50.486,-178.898,6.044,148.757
C04330=1187.373,95.930,-50.504,-178.896,6.044,148.756
C04331=1187.368,96.178,-50.522,-178.893,6.046,148.756
C04332=1187.363,96.428,-50.541,-178.891,6.047,148.755
C04333=1187.358,96.678,-50.559,-178.888,6.047,148.755
C04334=1187.353,96.927,-50.577,-178.885,6.049,148.754
C04335=1187.348,97.176,-50.595,-178.883,6.050,148.754
C04336=1187.344,97.425,-50.613,-178.880,6.051,148.753
C04337=1187.339,97.674,-50.631,-178.877,6.052,148.753
C04338=1187.334,97.924,-50.651,-178.875,6.054,148.752
C04339=1187.329,98.173,-50.669,-178.872,6.054,148.752
C04340=1187.324,98.422,-50.687,-178.869,6.056,148.751
C04341=1187.319,98.671,-50.705,-178.867,6.057,148.751
C04342=1187.315,98.921,-50.724,-178.864,6.058,148.750
C04343=1187.309,99.170,-50.742,-178.862,6.059,148.750
C04344=1187.305,99.419,-50.760,-178.859,6.061,148.749
C04345=1187.300,99.668,-50.778,-178.857,6.062,148.749
C04346=1187.295,99.918,-50.797,-178.853,6.063,148.748
C04347=1187.290,100.167,-50.816,-178.851,6.064,148.748
C04348=1187.285,100.416,-50.834,-178.849,6.066,148.747
C04349=1187.280,100.665,-50.852,-178.846,6.066,148.747
C04350=1187.276,100.915,-50.871,-178.843,6.068,148.746
C04351=1187.271,101.164,-50.890,-178.841,6.068,148.746
C04352=1187.266,101.413,-50.908,-178.838,6.070,148.745
C04353=1187.262,101.663,-50.927,-178.835,6.071,148.744
C04354=1187.257,101.912,-50.945,-178.833,6.072,148.744
C04355=1187.251,102.161,-50.963,-178.831,6.073,148.744
C04356=1187.247,102.411,-50.982,-178.827,6.075,148.743
C04357=1187.242,102.660,-51.000,-178.825,6.076,148.743
C04358=1187.236,102.909,-51.019,-178.822,6.077,148.742
C04359=1187.232,103.158,-51.037,-178.819,6.079,148.742
C04360=1187.228,103.408,-51.056,-178.817,6.079,148.741
C04361=1187.222,103.657,-51.075,-178.814,6.081,148.740
C04362=1187.217,103.906,-51.093,-178.812,6.082,148.740
C04363=1187.213,104.156,-51.111,-178.809,6.083,148.739
C04364=1187.208,104.404,-51.131,-178.806,6.084,148.739
C04365=1187.203,104.654,-51.149,-178.803,6.086,148.738
C04366=1187.198,104.903,-51.168,-178.801,6.087,148.738
C04367=1187.193,105.152,-51.186,-178.798,6.088,148.738
C04368=1187.189,105.402,-51.205,-178.796,6.089,148.737
C04369=1187.183,105.651,-51.224,-178.793,6.091,148.737
C04370=1187.179,105.900,-51.243,-178.791,6.091,148.736
C04371=1187.174,106.150,-51.262,-178.788,6.093,148.735
C04372=1187.169,106.418,-51.282,-178.785,6.094,148.735
C04373=1187.163,106.686,-51.302,-178.782,6.095,148.734
C04374=1187.159,106.955,-51.322,-178.779,6.097,148.734
C04375=1187.153,107.223,-51.342,-178.777,6.098,148.733
C04376=1187.148,107.472,-51.360,-178.774,6.099,148.733
C04377=1187.144,107.722,-51.380,-178.771,6.101,148.732
C04378=1187.139,107.970,-51.399,-178.768,6.102,148.732
C04379=1187.134,108.220,-51.418,-178.766,6.103,148.731
C04380=1187.129,108.469,-51.436,-178.763,6.105,148.731
C04381=1187.124,108.719,-51.455,-178.761,6.105,148.730
C04382=1187.120,108.968,-51.474,-178.758,6.107,148.730
C04383=1187.114,109.217,-51.493,-178.756,6.108,148.729
C04384=1187.110,109.467,-51.512,-178.753,6.109,148.729
C04385=1187.105,109.715,-51.531,-178.750,6.110,148.728
C04386=1187.101,109.965,-51.550,-178.747,6.112,148.728
C04387=1187.095,110.214,-51.568,-178.745,6.113,148.727
C04388=1187.090,110.463,-51.587,-178.742,6.114,148.727
C04389=1187.086,110.712,-51.607,-178.739,6.116,148.726
C04390=1187.081,110.961,-51.625,-178.737,6.117,148.726
C04391=1187.076,111.211,-51.644,-178.734,6.118,148.725
C04392=1187.071,111.460,-51.663,-178.732,6.119,148.725
C04393=1187.067,111.709,-51.683,-178.729,6.121,148.724
C04394=1187.061,111.959,-51.701,-178.726,6.122,148.724
C04395=1187.057,112.208,-51.720,-178.724,6.123,148.723
C04396=1187.052,112.457,-51.740,-178.721,6.125,148.723
C04397=1187.048,112.706,-51.759,-178.718,6.125,148.722
C04398=1187.042,112.955,-51.777,-178.716,6.127,148.722
C04399=1187.037,113.205,-51.797,-178.714,6.128,148.722
C04400=1187.033,113.454,-51.816,-178.710,6.129,148.721
C04401=1187.028,113.703,-51.835,-178.708,6.131,148.721
C04402=1187.023,113.952,-51.854,-178.705,6.132,148.720
C04403=1187.018,114.202,-51.873,-178.702,6.133,148.719
C04404=1187.013,114.451,-51.892,-178.700,6.134,148.719
C04405=1187.009,114.700,-51.911,-178.697,6.136,148.718
C04406=1187.004,114.949,-51.931,-178.694,6.137,148.718
C04407=1186.999,115.198,-51.950,-178.692,6.138,148.718
C04408=1186.994,115.447,-51.969,-178.689,6.140,148.717
C04409=1186.989,115.697,-51.989,-178.687,6.141,148.717
C04410=1186.984,115.946,-52.007,-178.684,6.142,148.716
C04411=1186.980,116.195,-52.026,-178.681,6.144,148.716
C04412=1186.975,116.445,-52.046,-178.679,6.145,148.715
C04413=1186.970,116.694,-52.065,-178.676,6.147,148.715
C04414=1186.965,116.943,-52.085,-178.674,6.147,148.714
C04415=1186.960,117.192,-52.104,-178.671,6.149,148.714
C04416=1186.956,117.441,-52.123,-178.668,6.151,148.713
C04417=1186.950,117.690,-52.143,-178.666,6.151,148.713
C04418=1186.946,117.940,-52.162,-178.663,6.153,148.712
C04419=1186.941,118.189,-52.181,-178.660,6.155,148.712
C04420=1186.936,118.438,-52.201,-178.658,6.155,148.711
C04421=1186.931,118.688,-52.220,-178.655,6.157,148.711
C04422=1186.927,118.936,-52.239,-178.653,6.158,148.710
C04423=1186.922,119.186,-52.259,-178.650,6.159,148.710
C04424=1186.917,119.435,-52.278,-178.647,6.161,148.709
C04425=1186.912,119.684,-52.297,-178.645,6.162,148.709
C04426=1186.907,119.934,-52.317,-178.642,6.163,148.708
C04427=1186.903,120.182,-52.336,-178.639,6.165,148.708
C04428=1186.898,120.432,-52.355,-178.637,6.166,148.708
C04429=1186.893,120.681,-52.375,-178.634,6.167,148.707
C04430=1186.888,120.930,-52.394,-178.631,6.168,148.707
C04431=1186.883,121.179,-52.415,-178.629,6.170,148.706
C04432=1186.879,121.428,-52.434,-178.626,6.172,148.706
C04433=1186.874,121.677,-52.453,-178.623,6.172,148.705
C04434=1186.869,121.927,-52.473,-178.621,6.174,148.705
C04435=1186.864,122.176,-52.492,-178.618,6.176,148.704
C04436=1186.859,122.425,-52.512,-178.615,6.177,148.704
C04437=1186.854,122.675,-52.531,-178.613,6.178,148.703
C04438=1186.849,122.923,-52.551,-178.610,6.180,148.703
C04439=1186.845,123.172,-52.570,-178.607,6.181,148.702
C04440=1186.841,123.422,-52.590,-178.605,6.182,148.702
C04441=1186.836,123.672,-52.610,-178.602,6.184,148.701
C04442=1186.831,123.920,-52.629,-178.599,6.185,148.701
C04443=1186.826,124.169,-52.649,-178.597,6.186,148.700
C04444=1186.821,124.419,-52.669,-178.594,6.188,148.700
C04445=1186.816,124.668,-52.688,-178.591,6.189,148.699
C04446=1186.811,124.917,-52.708,-178.589,6.191,148.699
C04447=1186.807,125.166,-52.728,-178.586,6.192,148.699
C04448=1186.802,125.415,-52.748,-178.583,6.193,148.698
C04449=1186.797,125.665,-52.767,-178.581,6.195,148.698
C04450=1186.792,125.914,-52.788,-178.578,6.196,148.697
C04451=1186.788,126.163,-52.807,-178.576,6.197,148.697
C04452=1186.783,126.412,-52.826,-178.573,6.199,148.696
C04453=1186.779,126.661,-52.846,-178.570,6.200,148.696
C04454=1186.774,126.910,-52.866,-178.568,6.201,148.695
C04455=1186.769,127.160,-52.886,-178.565,6.203,148.695
C04456=1186.764,127.408,-52.906,-178.562,6.205,148.694
C04457=1186.759,127.658,-52.925,-178.560,6.205,148.694
C04458=1186.755,127.907,-52.945,-178.557,6.207,148.694
C04459=1186.750,128.156,-52.965,-178.554,6.209,148.693
C04460=1186.745,128.405,-52.985,-178.552,6.210,148.693
C04461=1186.740,128.654,-53.005,-178.549,6.211,148.692
C04462=1186.736,128.904,-53.025,-178.546,6.213,148.692
C04463=1186.731,129.153,-53.044,-178.544,6.214,148.691
C04464=1186.726,129.402,-53.065,-178.541,6.215,148.691
C04465=1186.720,129.651,-53.085,-178.539,6.217,148.690
C04466=1186.716,129.900,-53.105,-178.536,6.218,148.690
C04467=1186.711,130.150,-53.125,-178.533,6.219,148.689
C04468=1186.707,130.399,-53.145,-178.531,6.221,148.689
C04469=1186.702,130.648,-53.165,-178.528,6.223,148.689
C04470=1186.697,130.897,-53.185,-178.525,6.224,148.688
C04471=1186.692,131.146,-53.204,-178.523,6.225,148.687
C04472=1186.688,131.395,-53.225,-178.520,6.227,148.687
C04473=1186.683,131.645,-53.244,-178.518,6.228,148.687
C04474=1186.678,131.894,-53.265,-178.515,6.229,148.686
C04475=1186.672,132.143,-53.285,-178.512,6.231,148.686
C04476=1186.668,132.412,-53.307,-178.509,6.233,148.685
C04477=1186.663,132.681,-53.329,-178.506,6.234,148.685
C04478=1186.658,132.949,-53.350,-178.503,6.236,148.684
C04479=1186.653,133.218,-53.372,-178.501,6.237,148.684
C04480=1186.648,133.466,-53.392,-178.498,6.238,148.683
C04481=1186.643,133.715,-53.412,-178.495,6.240,148.683
C04482=1186.638,133.964,-53.432,-178.493,6.242,148.683
C04483=1186.634,134.213,-53.452,-178.490,6.243,148.682
C04484=1186.628,134.463,-53.473,-178.487,6.244,148.681
C04485=1186.624,134.712,-53.493,-178.485,6.246,148.681
C04486=1186.620,134.961,-53.513,-178.482,6.248,148.681
C04487=1186.615,135.211,-53.533,-178.479,6.248,148.680
C04488=1186.610,135.460,-53.553,-178.477,6.250,148.680
C04489=1186.605,135.708,-53.574,-178.474,6.252,148.679
C04490=1186.600,135.958,-53.594,-178.472,6.253,148.679
C04491=1186.595,136.207,-53.614,-178.469,6.254,148.678
C04492=1186.591,136.456,-53.634,-178.466,6.256,148.678
C04493=1186.586,136.705,-53.655,-178.463,6.258,148.678
C04494=1186.581,136.954,-53.675,-178.461,6.259,148.677
C04495=1186.577,137.203,-53.695,-178.458,6.260,148.677
C04496=1186.571,137.453,-53.716,-178.455,6.262,148.676
C04497=1186.567,137.702,-53.737,-178.453,6.264,148.676
C04498=1186.562,137.951,-53.756,-178.450,6.265,148.675
C04499=1186.558,138.200,-53.777,-178.448,6.266,148.675
C04500=1186.553,138.449,-53.798,-178.445,6.268,148.674
C04501=1186.548,138.698,-53.818,-178.442,6.270,148.674
C04502=1186.544,138.947,-53.839,-178.440,6.270,148.674
C04503=1186.539,139.196,-53.860,-178.437,6.272,148.673
C04504=1186.533,139.445,-53.879,-178.434,6.274,148.673
C04505=1186.529,139.694,-53.899,-178.431,6.275,148.672
C04506=1186.524,139.944,-53.920,-178.429,6.276,148.672
C04507=1186.519,140.192,-53.941,-178.426,6.278,148.671
C04508=1186.515,140.441,-53.961,-178.424,6.280,148.671
C04509=1186.510,140.691,-53.982,-178.421,6.282,148.671
C04510=1186.505,140.940,-54.002,-178.418,6.283,148.670
C04511=1186.500,141.189,-54.023,-178.416,6.284,148.670
C04512=1186.496,141.438,-54.044,-178.413,6.286,148.669
C04513=1186.491,141.687,-54.064,-178.410,6.288,148.669
C04514=1186.486,141.936,-54.085,-178.408,6.289,148.668
C04515=1186.481,142.185,-54.105,-178.405,6.290,148.668
C04516=1186.476,142.434,-54.126,-178.402,6.292,148.667
C04517=1186.472,142.683,-54.147,-178.400,6.293,148.667
C04518=1186.468,142.933,-54.167,-178.397,6.295,148.667
C04519=1186.463,143.182,-54.188,-178.394,6.297,148.666
C04520=1186.458,143.431,-54.209,-178.392,6.298,148.666
C04521=1186.453,143.680,-54.230,-178.389,6.299,148.665
C04522=1186.449,143.929,-54.250,-178.386,6.301,148.665
C04523=1186.444,144.179,-54.271,-178.384,6.303,148.665
C04524=1186.439,144.427,-54.291,-178.382,6.304,148.664
C04525=1186.434,144.677,-54.312,-178.379,6.306,148.664
C04526=1186.430,144.926,-54.333,-178.376,6.307,148.663
C04527=1186.424,145.175,-54.354,-178.373,6.309,148.663
C04528=1186.420,145.424,-54.374,-178.370,6.310,148.662
C04529=1186.415,145.673,-54.395,-178.368,6.311,148.662
C04530=1186.411,145.921,-54.416,-178.365,6.313,148.662
C04531=1186.406,146.171,-54.437,-178.363,6.315,148.661
C04532=1186.401,146.420,-54.457,-178.360,6.316,148.661
C04533=1186.396,146.670,-54.479,-178.357,6.318,148.660
C04534=1186.392,146.919,-54.499,-178.354,6.320,148.660
C04535=1186.387,147.168,-54.520,-178.352,6.321,148.659
C04536=1186.383,147.416,-54.541,-178.349,6.323,148.659
C04537=1186.378,147.665,-54.562,-178.347,6.324,148.659
C04538=1186.372,147.915,-54.583,-178.344,6.326,148.658
C04539=1186.368,148.164,-54.603,-178.341,6.328,148.658
C04540=1186.363,148.412,-54.625,-178.339,6.328,148.657
C04541=1186.359,148.662,-54.646,-178.336,6.330,148.657
C04542=1186.354,148.911,-54.667,-178.333,6.332,148.657
C04543=1186.349,149.160,-54.688,-178.331,6.334,148.656
C04544=1186.345,149.409,-54.709,-178.328,6.335,148.656
C04545=1186.340,149.658,-54.730,-178.325,6.337,148.655
C04546=1186.334,149.907,-54.751,-178.323,6.338,148.655
C04547=1186.330,150.156,-54.772,-178.320,6.340,148.654
C04548=1186.326,150.406,-54.793,-178.317,6.341,148.654
C04549=1186.321,150.655,-54.814,-178.315,6.343,148.654
C04550=1186.316,150.903,-54.835,-178.312,6.345,148.653
C04551=1186.311,151.152,-54.856,-178.309,6.346,148.653
C04552=1186.306,151.402,-54.877,-178.307,6.347,148.652
C04553=1186.303,151.651,-54.899,-178.304,6.349,148.652
C04554=1186.297,151.900,-54.920,-178.301,6.351,148.652
C04555=1186.292,152.149,-54.941,-178.299,6.353,148.651
C04556=1186.288,152.398,-54.962,-178.296,6.354,148.651
C04557=1186.283,152.647,-54.983,-178.293,6.356,148.650
C04558=1186.279,152.896,-55.005,-178.291,6.357,148.650
C04559=1186.273,153.145,-55.026,-178.288,6.359,148.649
C04560=1186.269,153.394,-55.047,-178.285,6.360,148.649
C04561=1186.264,153.643,-55.068,-178.283,6.362,148.649
C04562=1186.259,153.892,-55.089,-178.280,6.364,148.648
C04563=1186.255,154.142,-55.111,-178.277,6.366,148.648
C04564=1186.250,154.391,-55.131,-178.275,6.367,148.648
C04565=1186.245,154.639,-55.153,-178.272,6.368,148.647
C04566=1186.240,154.889,-55.174,-178.270,6.370,148.647
C04567=1186.236,155.138,-55.196,-178.267,6.372,148.646
C04568=1186.231,155.386,-55.218,-178.264,6.373,148.646
C04569=1186.227,155.635,-55.238,-178.261,6.375,148.645
C04570=1186.222,155.884,-55.260,-178.259,6.377,148.645
C04571=1186.217,156.134,-55.281,-178.256,6.379,148.645
C04572=1186.212,156.383,-55.303,-178.253,6.380,148.644
C04573=1186.207,156.632,-55.324,-178.251,6.381,148.644
C04574=1186.204,156.881,-55.345,-178.248,6.383,148.643
C04575=1186.199,157.130,-55.367,-178.246,6.385,148.643
C04576=1186.194,157.379,-55.388,-178.243,6.387,148.643
C04577=1186.189,157.628,-55.409,-178.240,6.388,148.642
C04578=1186.184,157.877,-55.431,-178.237,6.390,148.642
C04579=1186.179,158.126,-55.452,-178.235,6.392,148.641
C04580=1186.175,158.395,-55.475,-178.232,6.393,148.641
C04581=1186.169,158.664,-55.499,-178.229,6.395,148.641
C04582=1186.165,158.933,-55.522,-178.226,6.397,148.640
C04583=1186.159,159.202,-55.545,-178.223,6.398,148.640
C04584=1186.154,159.451,-55.567,-178.221,6.400,148.639
C04585=1186.149,159.700,-55.589,-178.218,6.402,148.639
C04586=1186.145,159.950,-55.610,-178.215,6.404,148.639
C04587=1186.141,160.198,-55.631,-178.213,6.405,148.638
C04588=1186.136,160.447,-55.653,-178.210,6.407,148.638
C04589=1186.132,160.696,-55.675,-178.207,6.409,148.637
C04590=1186.127,160.945,-55.697,-178.205,6.410,148.637
C04591=1186.122,161.194,-55.718,-178.202,6.412,148.637
C04592=1186.117,161.443,-55.740,-178.200,6.414,148.636
C04593=1186.112,161.692,-55.761,-178.197,6.415,148.636
C04594=1186.108,161.941,-55.783,-178.194,6.417,148.636
C04595=1186.103,162.190,-55.805,-178.192,6.419,148.635
C04596=1186.099,162.440,-55.826,-178.189,6.420,148.635
C04597=1186.094,162.688,-55.848,-178.186,6.422,148.634
C04598=1186.089,162.937,-55.870,-178.183,6.424,148.634
C04599=1186.085,163.186,-55.892,-178.181,6.426,148.634
C04600=1186.080,163.435,-55.913,-178.178,6.427,148.633
C04601=1186.075,163.684,-55.935,-178.175,6.429,148.633
C04602=1186.071,163.933,-55.957,-178.173,6.430,148.632
C04603=1186.066,164.182,-55.979,-178.170,6.432,148.632
C04604=1186.061,164.431,-56.001,-178.168,6.434,148.632
C04605=1186.056,164.680,-56.023,-178.165,6.435,148.631
C04606=1186.051,164.930,-56.044,-178.162,6.437,148.631
C04607=1186.046,165.178,-56.066,-178.160,6.439,148.631
C04608=1186.042,165.428,-56.088,-178.157,6.441,148.630
C04609=1186.037,165.676,-56.110,-178.154,6.443,148.630
C04610=1186.033,165.926,-56.132,-178.152,6.444,148.629
C04611=1186.028,166.174,-56.154,-178.149,6.446,148.629
C04612=1186.023,166.423,-56.175,-178.146,6.448,148.629
C04613=1186.019,166.672,-56.197,-178.144,6.450,148.628
C04614=1186.014,166.920,-56.220,-178.141,6.451,148.628
C04615=1186.009,167.170,-56.242,-178.138,6.453,148.628
C04616=1186.005,167.419,-56.264,-178.136,6.455,148.627
C04617=1186.000,167.668,-56.286,-178.133,6.457,148.627
C04618=1185.995,167.917,-56.308,-178.131,6.458,148.626
C04619=1185.991,168.166,-56.330,-178.128,6.460,148.626
C04620=1185.986,168.415,-56.352,-178.125,6.461,148.625
C04621=1185.981,168.664,-56.374,-178.122,6.463,148.625
C04622=1185.976,168.913,-56.396,-178.120,6.465,148.625
C04623=1185.972,169.162,-56.418,-178.117,6.466,148.624
C04624=1185.968,169.410,-56.440,-178.114,6.468,148.624
C04625=1185.963,169.660,-56.463,-178.112,6.470,148.624
C04626=1185.958,169.909,-56.485,-178.109,6.472,148.623
C04627=1185.953,170.158,-56.507,-178.106,6.473,148.623
C04628=1185.949,170.407,-56.528,-178.104,6.475,148.623
C04629=1185.944,170.656,-56.550,-178.101,6.477,148.622
C04630=1185.940,170.905,-56.574,-178.098,6.479,148.622
C04631=1185.935,171.154,-56.595,-178.095,6.481,148.621
C04632=1185.930,171.403,-56.618,-178.093,6.482,148.621
C04633=1185.925,171.652,-56.640,-178.090,6.484,148.621
C04634=1185.921,171.901,-56.663,-178.087,6.486,148.620
C04635=1185.916,172.149,-56.684,-178.085,6.488,148.620
C04636=1185.912,172.399,-56.706,-178.082,6.489,148.620
C04637=1185.907,172.648,-56.729,-178.079,6.491,148.619
C04638=1185.902,172.896,-56.751,-178.077,6.493,148.619
C04639=1185.898,173.146,-56.773,-178.074,6.495,148.619
C04640=1185.892,173.395,-56.796,-178.071,6.497,148.618
C04641=1185.888,173.643,-56.818,-178.069,6.498,148.618
C04642=1185.884,173.892,-56.840,-178.066,6.500,148.617
C04643=1185.878,174.142,-56.863,-178.064,6.502,148.617
C04644=1185.875,174.390,-56.885,-178.061,6.504,148.617
C04645=1185.870,174.639,-56.907,-178.059,6.506,148.617
C04646=1185.865,174.888,-56.931,-178.056,6.508,148.616
C04647=1185.861,175.137,-56.953,-178.053,6.509,148.616
C04648=1185.855,175.386,-56.975,-178.050,6.511,148.616
C04649=1185.851,175.635,-56.998,-178.048,6.513,148.615
C04650=1185.846,175.884,-57.019,-178.045,6.515,148.615
C04651=1185.842,176.133,-57.043,-178.042,6.517,148.614
C04652=1185.837,176.382,-57.065,-178.040,6.518,148.614
C04653=1185.832,176.630,-57.088,-178.037,6.520,148.614
C04654=1185.828,176.880,-57.110,-178.034,6.522,148.613
C04655=1185.823,177.129,-57.133,-178.032,6.524,148.613
C04656=1185.818,177.377,-57.155,-178.029,6.525,148.613
C04657=1185.814,177.626,-57.178,-178.026,6.527,148.612
C04658=1185.809,177.876,-57.200,-178.024,6.529,148.612
C04659=1185.805,178.124,-57.223,-178.021,6.531,148.612
C04660=1185.800,178.373,-57.245,-178.018,6.533,148.611
C04661=1185.796,178.622,-57.268,-178.016,6.534,148.611
C04662=1185.791,178.872,-57.291,-178.013,6.536,148.610
C04663=1185.786,179.120,-57.313,-178.010,6.538,148.610
C04664=1185.781,179.369,-57.336,-178.008,6.540,148.610
C04665=1185.777,179.618,-57.358,-178.005,6.542,148.609
C04666=1185.772,179.867,-57.381,-178.002,6.543,148.609
C04667=1185.768,180.116,-57.404,-178.000,6.545,148.609
C04668=1185.763,180.365,-57.427,-177.998,6.547,148.609
C04669=1185.759,180.614,-57.450,-177.995,6.549,148.608
C04670=1185.753,180.863,-57.472,-177.992,6.551,148.608
C04671=1185.749,181.112,-57.495,-177.989,6.553,148.607
C04672=1185.745,181.360,-57.518,-177.987,6.554,148.607
C04673=1185.740,181.610,-57.541,-177.984,6.556,148.607
C04674=1185.735,181.858,-57.563,-177.981,6.559,148.606
C04675=1185.730,182.107,-57.586,-177.978,6.561,148.606
C04676=1185.726,182.356,-57.608,-177.976,6.562,148.606
C04677=1185.721,182.605,-57.632,-177.973,6.564,148.605
C04678=1185.716,182.854,-57.655,-177.970,6.566,148.605
C04679=1185.712,183.102,-57.678,-177.968,6.568,148.605
C04680=1185.707,183.351,-57.701,-177.965,6.569,148.604
C04681=1185.703,183.601,-57.723,-177.963,6.572,148.604
C04682=1185.698,183.850,-57.746,-177.960,6.573,148.604
C04683=1185.693,184.098,-57.769,-177.957,6.575,148.603
C04684=1185.689,184.368,-57.794,-177.955,6.577,148.603
C04685=1185.683,184.637,-57.819,-177.951,6.580,148.603
C04686=1185.678,184.907,-57.844,-177.949,6.581,148.602
C04687=1185.673,185.177,-57.868,-177.946,6.583,148.602
C04688=1185.669,185.426,-57.892,-177.943,6.585,148.602
C04689=1185.664,185.675,-57.915,-177.941,6.587,148.601
C04690=1185.660,185.923,-57.938,-177.938,6.589,148.601
C04691=1185.655,186.172,-57.961,-177.935,6.591,148.601
C04692=1185.651,186.421,-57.984,-177.932,6.593,148.600
C04693=1185.645,186.670,-58.007,-177.930,6.595,148.600
C04694=1185.641,186.919,-58.030,-177.927,6.597,148.600
C04695=1185.636,187.168,-58.053,-177.924,6.598,148.599
C04696=1185.632,187.417,-58.076,-177.922,6.600,148.599
C04697=1185.628,187.666,-58.099,-177.919,6.602,148.599
C04698=1185.623,187.915,-58.122,-177.917,6.604,148.598
C04699=1185.618,188.164,-58.146,-177.914,6.606,148.598
C04700=1185.614,188.413,-58.169,-177.911,6.608,148.598
C04701=1185.608,188.661,-58.192,-177.908,6.610,148.597
C04702=1185.604,188.910,-58.215,-177.905,6.612,148.597
C04703=1185.600,189.159,-58.238,-177.903,6.614,148.597
C04704=1185.595,189.408,-58.262,-177.900,6.616,148.596
C04705=1185.591,189.657,-58.286,-177.898,6.618,148.596
C04706=1185.586,189.906,-58.309,-177.895,6.620,148.596
C04707=1185.581,190.155,-58.332,-177.893,6.621,148.595
C04708=1185.577,190.403,-58.355,-177.890,6.623,148.595
C04709=1185.572,190.652,-58.378,-177.887,6.625,148.595
C04710=1185.568,190.901,-58.402,-177.885,6.627,148.594
C04711=1185.562,191.150,-58.425,-177.881,6.629,148.594
C04712=1185.558,191.399,-58.448,-177.879,6.631,148.594
C04713=1185.553,191.648,-58.472,-177.876,6.633,148.594
C04714=1185.549,191.896,-58.496,-177.874,6.635,148.593
C04715=1185.544,192.145,-58.519,-177.871,6.637,148.593
C04716=1185.540,192.394,-58.542,-177.868,6.639,148.593
C04717=1185.535,192.643,-58.565,-177.866,6.640,148.592
C04718=1185.531,192.892,-58.588,-177.863,6.642,148.592
C04719=1185.526,193.141,-58.612,-177.860,6.645,148.592
C04720=1185.521,193.389,-58.636,-177.858,6.647,148.591
C04721=1185.517,193.639,-58.659,-177.855,6.649,148.591
C04722=1185.512,193.888,-58.683,-177.852,6.651,148.591
C04723=1185.507,194.137,-58.706,-177.850,6.652,148.590
C04724=1185.503,194.385,-58.730,-177.847,6.654,148.590
C04725=1185.498,194.634,-58.753,-177.845,6.656,148.590
C04726=1185.494,194.883,-58.777,-177.842,6.658,148.589
C04727=1185.489,195.131,-58.801,-177.839,6.661,148.589
C04728=1185.485,195.380,-58.824,-177.836,6.662,148.589
C04729=1185.480,195.630,-58.848,-177.834,6.664,148.588
C04730=1185.475,195.878,-58.872,-177.831,6.666,148.588
C04731=1185.471,196.127,-58.895,-177.829,6.668,148.588
C04732=1185.466,196.376,-58.918,-177.826,6.670,148.588
C04733=1185.462,196.624,-58.942,-177.823,6.672,148.587
C04734=1185.457,196.873,-58.966,-177.820,6.674,148.587
C04735=1185.452,197.122,-58.989,-177.818,6.676,148.587
C04736=1185.448,197.371,-59.013,-177.815,6.678,148.586
C04737=1185.443,197.620,-59.037,-177.813,6.680,148.586
C04738=1185.439,197.868,-59.061,-177.810,6.682,148.586
C04739=1185.434,198.117,-59.084,-177.807,6.684,148.585
C04740=1185.430,198.366,-59.108,-177.804,6.686,148.585
C04741=1185.426,198.616,-59.132,-177.801,6.688,148.585
C04742=1185.420,198.864,-59.156,-177.799,6.690,148.585
C04743=1185.416,199.113,-59.180,-177.797,6.692,148.584
C04744=1185.411,199.362,-59.203,-177.794,6.694,148.584
C04745=1185.407,199.611,-59.227,-177.791,6.696,148.584
C04746=1185.402,199.859,-59.251,-177.788,6.698,148.583
C04747=1185.398,200.108,-59.275,-177.786,6.700,148.583
C04748=1185.393,200.357,-59.299,-177.783,6.702,148.583
C04749=1185.388,200.606,-59.322,-177.781,6.704,148.582
C04750=1185.383,200.854,-59.347,-177.778,6.706,148.582
C04751=1185.379,201.104,-59.371,-177.776,6.708,148.582
C04752=1185.375,201.352,-59.395,-177.773,6.711,148.582
C04753=1185.370,201.601,-59.419,-177.770,6.712,148.581
C04754=1185.366,201.850,-59.442,-177.767,6.714,148.581
C04755=1185.361,202.099,-59.467,-177.765,6.716,148.581
C04756=1185.356,202.348,-59.490,-177.762,6.718,148.581
C04757=1185.351,202.596,-59.514,-177.759,6.721,148.580
C04758=1185.348,202.845,-59.539,-177.756,6.723,148.580
C04759=1185.343,203.094,-59.562,-177.754,6.724,148.580
C04760=1185.338,203.343,-59.587,-177.752,6.726,148.579
C04761=1185.333,203.591,-59.611,-177.749,6.728,148.579
C04762=1185.329,203.840,-59.634,-177.746,6.731,148.579
C04763=1185.325,204.090,-59.658,-177.743,6.733,148.578
C04764=1185.320,204.338,-59.683,-177.740,6.735,148.578
C04765=1185.315,204.587,-59.707,-177.738,6.737,148.578
C04766=1185.311,204.836,-59.731,-177.736,6.738,148.578
C04767=1185.306,205.084,-59.755,-177.732,6.741,148.577
C04768=1185.301,205.333,-59.779,-177.730,6.743,148.577
C04769=1185.297,205.582,-59.804,-177.727,6.745,148.577
C04770=1185.293,205.830,-59.828,-177.725,6.747,148.576
C04771=1185.288,206.080,-59.852,-177.722,6.749,148.576
C04772=1185.283,206.328,-59.876,-177.719,6.751,148.576
C04773=1185.279,206.577,-59.900,-177.717,6.753,148.576
C04774=1185.274,206.826,-59.925,-177.714,6.755,148.575
C04775=1185.270,207.074,-59.949,-177.711,6.757,148.575
C04776=1185.265,207.323,-59.974,-177.708,6.760,148.575
C04777=1185.261,207.573,-59.997,-177.706,6.762,148.575
C04778=1185.256,207.821,-60.022,-177.703,6.764,148.574
C04779=1185.251,208.070,-60.046,-177.701,6.765,148.574
C04780=1185.247,208.318,-60.070,-177.699,6.767,148.574
C04781=1185.243,208.567,-60.095,-177.695,6.770,148.573
C04782=1185.238,208.816,-60.119,-177.693,6.772,148.573
C04783=1185.233,209.065,-60.143,-177.690,6.774,148.573
C04784=1185.228,209.313,-60.168,-177.688,6.776,148.573
C04785=1185.224,209.562,-60.193,-177.685,6.778,148.572
C04786=1185.219,209.811,-60.217,-177.682,6.780,148.572
C04787=1185.215,210.060,-60.241,-177.679,6.782,148.572
C04788=1185.210,210.330,-60.268,-177.677,6.785,148.572
C04789=1185.205,210.601,-60.295,-177.674,6.787,148.571
C04790=1185.200,210.871,-60.321,-177.671,6.789,148.571
C04791=1185.195,211.142,-60.348,-177.668,6.791,148.571
C04792=1185.191,211.391,-60.372,-177.665,6.794,148.570
C04793=1185.186,211.639,-60.397,-177.663,6.796,148.570
C04794=1185.181,211.888,-60.421,-177.660,6.798,148.570
C04795=1185.177,212.137,-60.446,-177.657,6.800,148.569
C04796=1185.173,212.385,-60.471,-177.654,6.802,148.569
C04797=1185.168,212.634,-60.495,-177.652,6.804,148.569
C04798=1185.164,212.883,-60.520,-177.649,6.806,148.569
C04799=1185.159,213.132,-60.545,-177.647,6.808,148.568
C04800=1185.154,213.380,-60.569,-177.644,6.811,148.568
C04801=1185.150,213.629,-60.594,-177.641,6.813,148.568
C04802=1185.145,213.878,-60.618,-177.638,6.815,148.568
C04803=1185.141,214.127,-60.644,-177.636,6.817,148.568
C04804=1185.136,214.375,-60.668,-177.633,6.819,148.567
C04805=1185.132,214.624,-60.692,-177.630,6.821,148.567
C04806=1185.127,214.873,-60.717,-177.628,6.823,148.567
C04807=1185.123,215.121,-60.742,-177.625,6.826,148.566
C04808=1185.118,215.370,-60.767,-177.622,6.828,148.566
C04809=1185.113,215.619,-60.792,-177.620,6.830,148.566
C04810=1185.109,215.868,-60.816,-177.618,6.832,148.566
C04811=1185.105,216.116,-60.842,-177.614,6.834,148.565
C04812=1185.100,216.365,-60.866,-177.612,6.836,148.565
C04813=1185.096,216.614,-60.891,-177.609,6.838,148.565
C04814=1185.091,216.862,-60.916,-177.606,6.841,148.565
C04815=1185.087,217.111,-60.940,-177.604,6.843,148.564
C04816=1185.082,217.360,-60.965,-177.601,6.845,148.564
C04817=1185.077,217.608,-60.991,-177.599,6.847,148.564
C04818=1185.073,217.857,-61.015,-177.596,6.849,148.564
C04819=1185.068,218.106,-61.040,-177.593,6.851,148.563
C04820=1185.064,218.355,-61.065,-177.591,6.853,148.563
C04821=1185.059,218.604,-61.090,-177.588,6.856,148.563
C04822=1185.055,218.853,-61.115,-177.585,6.858,148.563
C04823=1185.050,219.101,-61.140,-177.583,6.860,148.562
C04824=1185.046,219.350,-61.165,-177.580,6.862,148.562
C04825=1185.041,219.598,-61.190,-177.577,6.865,148.562
C04826=1185.037,219.847,-61.215,-177.575,6.866,148.562
C04827=1185.032,220.096,-61.240,-177.572,6.869,148.561
C04828=1185.028,220.345,-61.265,-177.569,6.871,148.561
C04829=1185.023,220.593,-61.291,-177.567,6.873,148.561
C04830=1185.019,220.842,-61.315,-177.564,6.875,148.561
C04831=1185.014,221.090,-61.340,-177.561,6.878,148.560
C04832=1185.010,221.340,-61.366,-177.559,6.880,148.560
C04833=1185.005,221.588,-61.391,-177.556,6.882,148.560
C04834=1185.000,221.837,-61.416,-177.553,6.884,148.560
C04835=1184.996,222.085,-61.441,-177.551,6.887,148.560
C04836=1184.992,222.334,-61.466,-177.548,6.888,148.559
C04837=1184.987,222.583,-61.491,-177.545,6.891,148.559
C04838=1184.983,222.831,-61.517,-177.543,6.893,148.559
C04839=1184.978,223.080,-61.542,-177.540,6.895,148.558
C04840=1184.973,223.329,-61.567,-177.537,6.898,148.558
C04841=1184.969,223.577,-61.592,-177.535,6.900,148.558
C04842=1184.965,223.826,-61.617,-177.532,6.902,148.558
C04843=1184.961,224.075,-61.643,-177.529,6.905,148.558
C04844=1184.956,224.323,-61.668,-177.527,6.906,148.557
C04845=1184.951,224.572,-61.693,-177.525,6.908,148.557
C04846=1184.946,224.821,-61.719,-177.521,6.911,148.557
C04847=1184.942,225.069,-61.744,-177.519,6.913,148.557
C04848=1184.937,225.318,-61.769,-177.517,6.915,148.556
C04849=1184.933,225.567,-61.795,-177.513,6.918,148.556
C04850=1184.929,225.816,-61.821,-177.511,6.920,148.556
C04851=1184.924,226.064,-61.846,-177.509,6.922,148.556
C04852=1184.919,226.313,-61.871,-177.505,6.924,148.555
C04853=1184.915,226.562,-61.897,-177.503,6.926,148.555
C04854=1184.910,226.810,-61.922,-177.500,6.928,148.555
C04855=1184.906,227.059,-61.948,-177.498,6.931,148.555
C04856=1184.901,227.307,-61.973,-177.495,6.933,148.555
C04857=1184.897,227.557,-61.998,-177.493,6.935,148.554
C04858=1184.892,227.805,-62.024,-177.490,6.938,148.554
C04859=1184.888,228.053,-62.049,-177.487,6.940,148.554
C04860=1184.883,228.302,-62.075,-177.485,6.942,148.554
C04861=1184.879,228.551,-62.101,-177.482,6.944,148.553
C04862=1184.874,228.799,-62.126,-177.479,6.947,148.553
C04863=1184.870,229.048,-62.152,-177.476,6.949,148.553
C04864=1184.866,229.297,-62.177,-177.474,6.951,148.553
C04865=1184.861,229.545,-62.203,-177.471,6.953,148.553
C04866=1184.856,229.794,-62.228,-177.469,6.956,148.553
C04867=1184.852,230.043,-62.254,-177.466,6.958,148.552
C04868=1184.847,230.291,-62.279,-177.463,6.960,148.552
C04869=1184.843,230.540,-62.305,-177.461,6.963,148.552
C04870=1184.839,230.789,-62.331,-177.458,6.965,148.551
C04871=1184.834,231.037,-62.356,-177.455,6.968,148.551
C04872=1184.830,231.286,-62.382,-177.453,6.969,148.551
C04873=1184.825,231.535,-62.408,-177.450,6.972,148.551
C04874=1184.821,231.784,-62.434,-177.447,6.974,148.551
C04875=1184.816,232.032,-62.460,-177.445,6.976,148.551
C04876=1184.812,232.281,-62.485,-177.442,6.978,148.550
C04877=1184.807,232.529,-62.511,-177.440,6.981,148.550
C04878=1184.803,232.778,-62.537,-177.437,6.983,148.550
C04879=1184.799,233.026,-62.563,-177.434,6.986,148.550
C04880=1184.794,233.275,-62.589,-177.432,6.988,148.549
C04881=1184.790,233.524,-62.615,-177.429,6.990,148.549
C04882=1184.785,233.772,-62.641,-177.426,6.992,148.549
C04883=1184.780,234.020,-62.666,-177.424,6.995,148.549
C04884=1184.776,234.269,-62.692,-177.421,6.997,148.549
C04885=1184.771,234.518,-62.718,-177.419,6.999,148.549
C04886=1184.767,234.767,-62.745,-177.416,7.001,148.548
C04887=1184.763,235.015,-62.770,-177.413,7.004,148.548
C04888=1184.758,235.263,-62.796,-177.411,7.006,148.548
C04889=1184.753,235.513,-62.822,-177.408,7.009,148.548
C04890=1184.749,235.761,-62.848,-177.405,7.011,148.547
C04891=1184.745,236.010,-62.874,-177.403,7.013,148.547
C04892=1184.740,236.281,-62.902,-177.400,7.016,148.547
C04893=1184.734,236.553,-62.931,-177.397,7.019,148.547
C04894=1184.730,236.824,-62.959,-177.394,7.021,148.547
C04895=1184.725,237.096,-62.987,-177.391,7.023,148.546
C04896=1184.721,237.345,-63.015,-177.389,7.026,148.546
C04897=1184.716,237.593,-63.040,-177.386,7.028,148.546
C04898=1184.712,237.842,-63.066,-177.383,7.031,148.546
C04899=1184.707,238.090,-63.093,-177.381,7.033,148.546
C04900=1184.703,238.339,-63.118,-177.378,7.036,148.546
C04901=1184.699,238.588,-63.144,-177.376,7.038,148.545
C04902=1184.694,238.836,-63.171,-177.373,7.040,148.545
C04903=1184.690,239.085,-63.197,-177.370,7.043,148.545
C04904=1184.685,239.332,-63.223,-177.368,7.044,148.545
C04905=1184.680,239.582,-63.250,-177.365,7.047,148.545
C04906=1184.676,239.830,-63.275,-177.362,7.049,148.544
C04907=1184.672,240.079,-63.302,-177.359,7.052,148.544
C04908=1184.667,240.328,-63.328,-177.357,7.054,148.544
C04909=1184.663,240.576,-63.355,-177.355,7.056,148.544
C04910=1184.658,240.825,-63.381,-177.352,7.059,148.544
C04911=1184.654,241.073,-63.407,-177.349,7.061,148.543
C04912=1184.649,241.322,-63.434,-177.347,7.064,148.543
C04913=1184.645,241.570,-63.460,-177.344,7.066,148.543
C04914=1184.640,241.819,-63.486,-177.341,7.069,148.543
C04915=1184.636,242.067,-63.513,-177.339,7.071,148.543
C04916=1184.632,242.316,-63.538,-177.336,7.074,148.543
C04917=1184.627,242.564,-63.565,-177.334,7.076,148.543
C04918=1184.623,242.813,-63.591,-177.330,7.078,148.542
C04919=1184.618,243.062,-63.618,-177.328,7.080,148.542
C04920=1184.614,243.310,-63.645,-177.325,7.083,148.542
C04921=1184.609,243.559,-63.671,-177.323,7.085,148.542
C04922=1184.605,243.807,-63.698,-177.321,7.087,148.542
C04923=1184.600,244.056,-63.724,-177.317,7.090,148.541
C04924=1184.597,244.304,-63.750,-177.315,7.092,148.541
C04925=1184.592,244.553,-63.777,-177.312,7.095,148.541
C04926=1184.587,244.802,-63.804,-177.310,7.097,148.541
C04927=1184.583,245.050,-63.830,-177.307,7.100,148.541
C04928=1184.578,245.299,-63.857,-177.305,7.102,148.541
C04929=1184.574,245.548,-63.883,-177.302,7.105,148.540
C04930=1184.569,245.796,-63.910,-177.299,7.107,148.540
C04931=1184.566,246.044,-63.937,-177.296,7.110,148.540
C04932=1184.561,246.293,-63.964,-177.294,7.112,148.540
C04933=1184.556,246.542,-63.990,-177.291,7.114,148.540
C04934=1184.552,246.790,-64.016,-177.289,7.117,148.540
C04935=1184.547,247.038,-64.043,-177.286,7.120,148.540
C04936=1184.543,247.287,-64.070,-177.284,7.121,148.539
C04937=1184.538,247.536,-64.096,-177.281,7.124,148.539
C04938=1184.534,247.784,-64.123,-177.279,7.126,148.539
C04939=1184.530,248.032,-64.150,-177.275,7.129,148.539
C04940=1184.525,248.281,-64.177,-177.273,7.131,148.539
C04941=1184.521,248.529,-64.204,-177.270,7.134,148.538
C04942=1184.517,248.778,-64.230,-177.268,7.136,148.538
C04943=1184.512,249.027,-64.257,-177.265,7.139,148.538
C04944=1184.507,249.275,-64.284,-177.263,7.141,148.538
C04945=1184.502,249.524,-64.311,-177.260,7.144,148.538
C04946=1184.498,249.772,-64.337,-177.258,7.146,148.538
C04947=1184.494,250.020,-64.364,-177.254,7.149,148.538
C04948=1184.489,250.269,-64.391,-177.252,7.151,148.537
C04949=1184.486,250.518,-64.418,-177.249,7.154,148.537
C04950=1184.481,250.766,-64.445,-177.247,7.156,148.537
C04951=1184.476,251.015,-64.472,-177.244,7.159,148.537
C04952=1184.472,251.263,-64.499,-177.242,7.161,148.537
C04953=1184.468,251.511,-64.526,-177.239,7.163,148.537
C04954=1184.463,251.760,-64.553,-177.237,7.166,148.537
C04955=1184.459,252.008,-64.580,-177.234,7.169,148.536
C04956=1184.454,252.257,-64.607,-177.231,7.170,148.536
C04957=1184.449,252.505,-64.634,-177.228,7.173,148.536
C04958=1184.446,252.754,-64.661,-177.226,7.176,148.536
C04959=1184.441,253.003,-64.688,-177.224,7.179,148.536
C04960=1184.437,253.251,-64.715,-177.220,7.181,148.536
C04961=1184.432,253.500,-64.742,-177.218,7.183,148.536
C04962=1184.427,253.748,-64.769,-177.215,7.186,148.536
C04963=1184.423,253.997,-64.796,-177.213,7.188,148.535
C04964=1184.420,254.245,-64.824,-177.210,7.191,148.535
C04965=1184.415,254.494,-64.851,-177.208,7.193,148.535
C04966=1184.410,254.742,-64.878,-177.205,7.196,148.535
C04967=1184.406,254.991,-64.905,-177.203,7.198,148.535
C04968=1184.401,255.239,-64.932,-177.200,7.201,148.535
C04969=1184.396,255.488,-64.959,-177.198,7.203,148.535
C04970=1184.393,255.736,-64.987,-177.194,7.206,148.534
C04971=1184.388,255.985,-65.014,-177.192,7.209,148.534
C04972=1184.383,256.233,-65.041,-177.190,7.211,148.534
C04973=1184.379,256.481,-65.068,-177.187,7.214,148.534
C04974=1184.375,256.729,-65.096,-177.184,7.216,148.534
C04975=1184.371,256.978,-65.123,-177.181,7.219,148.534
C04976=1184.366,257.227,-65.150,-177.179,7.221,148.534
C04977=1184.362,257.475,-65.177,-177.176,7.224,148.533
C04978=1184.357,257.723,-65.205,-177.173,7.227,148.533
C04979=1184.353,257.972,-65.232,-177.171,7.229,148.533
C04980=1184.349,258.221,-65.260,-177.168,7.232,148.533
C04981=1184.344,258.469,-65.287,-177.166,7.234,148.533
C04982=1184.340,258.717,-65.314,-177.163,7.237,148.533
C04983=1184.336,258.967,-65.342,-177.161,7.239,148.533
C04984=1184.331,259.214,-65.370,-177.158,7.242,148.533
C04985=1184.327,259.463,-65.397,-177.155,7.244,148.532
C04986=1184.322,259.711,-65.424,-177.153,7.246,148.532
C04987=1184.318,259.960,-65.452,-177.150,7.249,148.532
C04988=1184.313,260.208,-65.479,-177.148,7.252,148.532
C04989=1184.309,260.456,-65.507,-177.145,7.255,148.532
C04990=1184.305,260.706,-65.534,-177.143,7.256,148.532
C04991=1184.300,260.954,-65.562,-177.140,7.259,148.532
C04992=1184.295,261.202,-65.590,-177.137,7.262,148.532
C04993=1184.291,261.450,-65.617,-177.135,7.265,148.532
C04994=1184.287,261.699,-65.645,-177.132,7.267,148.531
C04995=1184.283,261.947,-65.672,-177.130,7.269,148.531
C04996=1184.278,262.221,-65.703,-177.127,7.272,148.531
C04997=1184.273,262.493,-65.733,-177.124,7.275,148.531
C04998=1184.269,262.766,-65.764,-177.121,7.278,148.531
C04999=1184.263,263.039,-65.794,-177.118,7.281,148.531
C05000=1184.259,263.288,-65.821,-177.115,7.284,148.531
C05001=1184.255,263.536,-65.849,-177.113,7.287,148.531
C05002=1184.250,263.785,-65.877,-177.110,7.289,148.530
C05003=1184.246,264.033,-65.905,-177.107,7.292,148.530
C05004=1184.242,264.281,-65.933,-177.105,7.294,148.530
C05005=1184.237,264.530,-65.960,-177.102,7.297,148.530
C05006=1184.233,264.778,-65.988,-177.100,7.300,148.530
C05007=1184.228,265.026,-66.016,-177.097,7.302,148.530
C05008=1184.223,265.275,-66.043,-177.094,7.305,148.530
C05009=1184.220,265.523,-66.071,-177.092,7.307,148.530
C05010=1184.215,265.771,-66.099,-177.090,7.310,148.530
C05011=1184.211,266.021,-66.127,-177.087,7.313,148.530
C05012=1184.206,266.269,-66.155,-177.084,7.315,148.529
C05013=1184.202,266.517,-66.183,-177.081,7.318,148.529
C05014=1184.198,266.765,-66.211,-177.079,7.321,148.529
C05015=1184.193,267.014,-66.239,-177.077,7.323,148.529
C05016=1184.189,267.263,-66.267,-177.074,7.326,148.529
C05017=1184.185,267.510,-66.295,-177.072,7.328,148.529
C05018=1184.179,267.759,-66.323,-177.069,7.331,148.529
C05019=1184.176,268.007,-66.351,-177.066,7.334,148.529
C05020=1184.171,268.255,-66.379,-177.064,7.336,148.529
C05021=1184.167,268.504,-66.406,-177.061,7.339,148.529
C05022=1184.162,268.752,-66.435,-177.058,7.342,148.529
C05023=1184.158,269.001,-66.463,-177.056,7.344,148.528
C05024=1184.153,269.249,-66.491,-177.053,7.347,148.528
C05025=1184.150,269.498,-66.519,-177.050,7.350,148.528
C05026=1184.145,269.746,-66.547,-177.048,7.352,148.528
C05027=1184.141,269.995,-66.576,-177.045,7.355,148.528
C05028=1184.136,270.242,-66.604,-177.042,7.358,148.528
C05029=1184.133,270.491,-66.632,-177.040,7.360,148.528
C05030=1184.128,270.739,-66.660,-177.037,7.363,148.528
C05031=1184.124,270.988,-66.687,-177.035,7.366,148.528
C05032=1184.118,271.237,-66.716,-177.033,7.368,148.528
C05033=1184.115,271.485,-66.744,-177.029,7.371,148.527
C05034=1184.110,271.733,-66.772,-177.027,7.374,148.527
C05035=1184.106,271.982,-66.801,-177.025,7.376,148.527
C05036=1184.102,272.229,-66.829,-177.022,7.379,148.527
C05037=1184.097,272.478,-66.858,-177.019,7.382,148.527
C05038=1184.093,272.726,-66.886,-177.017,7.384,148.527
C05039=1184.089,272.975,-66.914,-177.014,7.387,148.527
C05040=1184.084,273.223,-66.942,-177.011,7.390,148.527
C05041=1184.080,273.472,-66.971,-177.009,7.392,148.527
C05042=1184.075,273.719,-66.999,-177.006,7.395,148.527
C05043=1184.071,273.968,-67.027,-177.003,7.398,148.527
C05044=1184.067,274.217,-67.055,-177.001,7.400,148.527
C05045=1184.062,274.465,-67.084,-176.998,7.403,148.527
C05046=1184.059,274.713,-67.113,-176.996,7.406,148.527
C05047=1184.053,274.961,-67.141,-176.994,7.408,148.526
C05048=1184.050,275.210,-67.169,-176.991,7.411,148.526
C05049=1184.045,275.458,-67.198,-176.988,7.414,148.526
C05050=1184.041,275.707,-67.226,-176.986,7.416,148.526
C05051=1184.037,275.955,-67.255,-176.983,7.419,148.526
C05052=1184.032,276.203,-67.284,-176.981,7.422,148.526
C05053=1184.028,276.452,-67.312,-176.978,7.424,148.526
C05054=1184.023,276.700,-67.340,-176.975,7.427,148.526
C05055=1184.019,276.948,-67.369,-176.972,7.430,148.526
C05056=1184.015,277.197,-67.398,-176.970,7.433,148.526
C05057=1184.010,277.445,-67.426,-176.968,7.435,148.526
C05058=1184.006,277.693,-67.454,-176.965,7.438,148.526
C05059=1184.002,277.942,-67.484,-176.962,7.441,148.526
C05060=1183.997,278.190,-67.511,-176.960,7.443,148.526
C05061=1183.993,278.438,-67.540,-176.957,7.446,148.526
C05062=1183.989,278.687,-67.570,-176.955,7.449,148.526
C05063=1183.984,278.935,-67.597,-176.952,7.451,148.525
C05064=1183.980,279.183,-67.627,-176.950,7.454,148.525
C05065=1183.976,279.432,-67.656,-176.947,7.457,148.525
C05066=1183.971,279.680,-67.683,-176.944,7.460,148.525
C05067=1183.967,279.928,-67.713,-176.942,7.462,148.525
C05068=1183.963,280.177,-67.742,-176.939,7.465,148.525
C05069=1183.959,280.424,-67.770,-176.937,7.468,148.525
C05070=1183.954,280.673,-67.799,-176.934,7.471,148.525
C05071=1183.950,280.921,-67.828,-176.932,7.474,148.525
C05072=1183.945,281.169,-67.857,-176.929,7.477,148.525
C05073=1183.942,281.417,-67.885,-176.926,7.480,148.525
C05074=1183.937,281.666,-67.914,-176.924,7.482,148.525
C05075=1183.933,281.914,-67.944,-176.921,7.485,148.525
C05076=1183.928,282.163,-67.972,-176.919,7.488,148.525
C05077=1183.924,282.411,-68.001,-176.916,7.491,148.525
C05078=1183.920,282.659,-68.030,-176.914,7.493,148.525
C05079=1183.915,282.907,-68.059,-176.911,7.496,148.524
C05080=1183.911,283.155,-68.088,-176.908,7.499,148.524
C05081=1183.906,283.404,-68.117,-176.906,7.501,148.524
C05082=1183.902,283.652,-68.146,-176.903,7.504,148.524
C05083=1183.898,283.900,-68.174,-176.900,7.507,148.524
C05084=1183.894,284.149,-68.204,-176.897,7.510,148.524
C05085=1183.889,284.397,-68.233,-176.895,7.512,148.524
C05086=1183.885,284.646,-68.262,-176.893,7.515,148.524
C05087=1183.881,284.894,-68.291,-176.890,7.518,148.524
C05088=1183.876,285.142,-68.320,-176.888,7.521,148.524
C05089=1183.872,285.390,-68.349,-176.885,7.523,148.524
C05090=1183.867,285.639,-68.378,-176.883,7.526,148.524
C05091=1183.864,285.887,-68.407,-176.880,7.529,148.524
C05092=1183.860,286.135,-68.437,-176.877,7.532,148.524
C05093=1183.855,286.383,-68.465,-176.875,7.534,148.524
C05094=1183.850,286.631,-68.495,-176.872,7.537,148.524
C05095=1183.846,286.880,-68.524,-176.870,7.540,148.524
C05096=1183.842,287.128,-68.554,-176.867,7.543,148.524
C05097=1183.838,287.376,-68.583,-176.865,7.546,148.524
C05098=1183.833,287.624,-68.611,-176.862,7.549,148.524
C05099=1183.829,287.873,-68.641,-176.859,7.552,148.524
C05100=1183.825,288.147,-68.674,-176.857,7.555,148.524
C05101=1183.819,288.422,-68.706,-176.854,7.558,148.524
C05102=1183.815,288.697,-68.738,-176.851,7.561,148.524
C05103=1183.810,288.971,-68.771,-176.848,7.564,148.524
C05104=1183.806,289.219,-68.800,-176.846,7.567,148.524
C05105=1183.801,289.467,-68.830,-176.843,7.570,148.524
C05106=1183.797,289.716,-68.859,-176.840,7.573,148.524
C05107=1183.793,289.964,-68.889,-176.838,7.576,148.524
C05108=1183.789,290.213,-68.917,-176.835,7.578,148.524
C05109=1183.784,290.461,-68.947,-176.833,7.581,148.523
C05110=1183.780,290.709,-68.976,-176.830,7.584,148.523
C05111=1183.775,290.957,-69.005,-176.827,7.587,148.523
C05112=1183.771,291.205,-69.035,-176.825,7.590,148.523
C05113=1183.767,291.454,-69.064,-176.822,7.592,148.523
C05114=1183.762,291.702,-69.094,-176.820,7.595,148.523
C05115=1183.758,291.950,-69.124,-176.817,7.598,148.523
C05116=1183.754,292.198,-69.154,-176.814,7.601,148.523
C05117=1183.750,292.446,-69.183,-176.812,7.604,148.523
C05118=1183.746,292.695,-69.213,-176.810,7.606,148.523
C05119=1183.742,292.943,-69.242,-176.807,7.609,148.523
C05120=1183.737,293.191,-69.272,-176.804,7.612,148.523
C05121=1183.733,293.439,-69.301,-176.802,7.615,148.523
C05122=1183.728,293.688,-69.331,-176.799,7.617,148.523
C05123=1183.724,293.936,-69.361,-176.797,7.620,148.523
C05124=1183.720,294.184,-69.391,-176.794,7.623,148.523
C05125=1183.716,294.432,-69.420,-176.791,7.626,148.523
C05126=1183.712,294.680,-69.450,-176.789,7.629,148.523
C05127=1183.708,294.929,-69.479,-176.787,7.632,148.523
C05128=1183.703,295.177,-69.509,-176.784,7.635,148.523
C05129=1183.699,295.425,-69.539,-176.781,7.638,148.523
C05130=1183.695,295.673,-69.569,-176.779,7.641,148.523
C05131=1183.690,295.921,-69.598,-176.776,7.644,148.523
C05132=1183.686,296.170,-69.628,-176.774,7.646,148.523
C05133=1183.682,296.418,-69.658,-176.771,7.649,148.523
C05134=1183.678,296.666,-69.688,-176.768,7.652,148.523
C05135=1183.673,296.914,-69.717,-176.766,7.655,148.523
C05136=1183.669,297.162,-69.748,-176.763,7.658,148.523
C05137=1183.665,297.410,-69.778,-176.761,7.661,148.523
C05138=1183.660,297.659,-69.807,-176.759,7.663,148.523
C05139=1183.656,297.906,-69.837,-176.756,7.666,148.523
C05140=1183.652,298.155,-69.867,-176.753,7.669,148.523
C05141=1183.647,298.403,-69.897,-176.750,7.672,148.523
C05142=1183.644,298.651,-69.927,-176.748,7.676,148.523
C05143=1183.639,298.899,-69.957,-176.746,7.678,148.523
C05144=1183.635,299.147,-69.987,-176.743,7.681,148.523
C05145=1183.631,299.395,-70.017,-176.741,7.684,148.523
C05146=1183.626,299.644,-70.047,-176.738,7.687,148.523
C05147=1183.622,299.892,-70.077,-176.735,7.690,148.523
C05148=1183.617,300.140,-70.107,-176.732,7.693,148.523
C05149=1183.613,300.388,-70.137,-176.731,7.695,148.523
C05150=1183.609,300.637,-70.167,-176.728,7.698,148.523
C05151=1183.605,300.885,-70.198,-176.725,7.701,148.523
C05152=1183.601,301.133,-70.227,-176.723,7.704,148.523
C05153=1183.596,301.381,-70.258,-176.720,7.707,148.523
C05154=1183.592,301.629,-70.287,-176.718,7.711,148.523
C05155=1183.588,301.877,-70.317,-176.715,7.713,148.523
C05156=1183.583,302.125,-70.348,-176.713,7.716,148.523
C05157=1183.579,302.373,-70.378,-176.710,7.719,148.523
C05158=1183.575,302.622,-70.409,-176.707,7.722,148.523
C05159=1183.571,302.870,-70.438,-176.705,7.725,148.523
C05160=1183.566,303.118,-70.469,-176.702,7.728,148.523
C05161=1183.562,303.366,-70.499,-176.700,7.730,148.523
C05162=1183.557,303.614,-70.529,-176.697,7.733,148.523
C05163=1183.554,303.862,-70.559,-176.695,7.736,148.523
C05164=1183.549,304.110,-70.590,-176.692,7.740,148.523
C05165=1183.545,304.359,-70.620,-176.690,7.743,148.523
C05166=1183.541,304.607,-70.651,-176.687,7.746,148.523
C05167=1183.537,304.854,-70.681,-176.685,7.748,148.523
C05168=1183.532,305.103,-70.711,-176.682,7.751,148.523
C05169=1183.528,305.351,-70.741,-176.680,7.754,148.523
C05170=1183.524,305.599,-70.772,-176.677,7.757,148.523
C05171=1183.520,305.847,-70.803,-176.674,7.760,148.523
C05172=1183.516,306.095,-70.833,-176.672,7.763,148.523
C05173=1183.511,306.343,-70.863,-176.669,7.766,148.524
C05174=1183.507,306.591,-70.893,-176.667,7.769,148.524
C05175=1183.503,306.840,-70.925,-176.665,7.772,148.524
C05176=1183.498,307.088,-70.955,-176.662,7.775,148.524
C05177=1183.494,307.335,-70.985,-176.660,7.778,148.524
C05178=1183.489,307.584,-71.015,-176.657,7.781,148.524
C05179=1183.485,307.832,-71.046,-176.654,7.784,148.524
C05180=1183.482,308.080,-71.077,-176.651,7.787,148.524
C05181=1183.477,308.328,-71.108,-176.649,7.790,148.524
C05182=1183.473,308.576,-71.138,-176.647,7.792,148.524
C05183=1183.468,308.824,-71.168,-176.644,7.795,148.524
C05184=1183.464,309.072,-71.200,-176.642,7.798,148.524
C05185=1183.460,309.320,-71.230,-176.639,7.802,148.524
C05186=1183.456,309.568,-71.261,-176.637,7.805,148.524
C05187=1183.452,309.817,-71.292,-176.634,7.808,148.524
C05188=1183.447,310.065,-71.322,-176.632,7.811,148.524
C05189=1183.443,310.312,-71.353,-176.630,7.813,148.524
C05190=1183.439,310.560,-71.383,-176.627,7.816,148.524
C05191=1183.435,310.809,-71.415,-176.624,7.819,148.524
C05192=1183.430,311.057,-71.445,-176.622,7.822,148.524
C05193=1183.426,311.305,-71.475,-176.619,7.825,148.524
C05194=1183.422,311.553,-71.507,-176.616,7.828,148.524
C05195=1183.418,311.801,-71.537,-176.614,7.832,148.524
C05196=1183.413,312.049,-71.568,-176.611,7.835,148.524
C05197=1183.410,312.297,-71.599,-176.609,7.837,148.524
C05198=1183.405,312.545,-71.629,-176.607,7.840,148.525
C05199=1183.401,312.793,-71.661,-176.604,7.843,148.525
C05200=1183.397,313.041,-71.692,-176.602,7.846,148.525
C05201=1183.392,313.289,-71.723,-176.599,7.850,148.525
C05202=1183.388,313.537,-71.753,-176.597,7.853,148.525
C05203=1183.384,313.786,-71.784,-176.594,7.856,148.525
C05204=1183.379,314.062,-71.819,-176.591,7.859,148.525
C05205=1183.375,314.338,-71.854,-176.589,7.862,148.525
C05206=1183.370,314.615,-71.888,-176.586,7.866,148.525
C05207=1183.365,314.892,-71.923,-176.583,7.869,148.525
C05208=1183.361,315.140,-71.954,-176.581,7.872,148.525
C05209=1183.357,315.388,-71.985,-176.578,7.875,148.525
C05210=1183.353,315.636,-72.016,-176.575,7.878,148.525
C05211=1183.348,315.884,-72.046,-176.573,7.881,148.525
C05212=1183.344,316.132,-72.077,-176.570,7.884,148.525
C05213=1183.340,316.380,-72.109,-176.568,7.887,148.525
C05214=1183.336,316.628,-72.140,-176.566,7.890,148.525
C05215=1183.332,316.876,-72.171,-176.563,7.893,148.525
C05216=1183.327,317.124,-72.202,-176.561,7.896,148.526
C05217=1183.323,317.372,-72.233,-176.558,7.899,148.526
C05218=1183.319,317.620,-72.265,-176.555,7.902,148.526
C05219=1183.315,317.868,-72.296,-176.553,7.905,148.526
C05220=1183.310,318.116,-72.327,-176.550,7.908,148.526
C05221=1183.307,318.364,-72.359,-176.548,7.912,148.526
C05222=1183.302,318.612,-72.389,-176.546,7.915,148.526
C05223=1183.298,318.860,-72.421,-176.543,7.918,148.526
C05224=1183.294,319.108,-72.452,-176.541,7.920,148.526
C05225=1183.290,319.356,-72.484,-176.538,7.923,148.526
C05226=1183.285,319.604,-72.515,-176.536,7.927,148.526
C05227=1183.282,319.852,-72.546,-176.533,7.930,148.526
C05228=1183.277,320.100,-72.577,-176.531,7.933,148.526
C05229=1183.273,320.348,-72.609,-176.528,7.936,148.526
C05230=1183.269,320.596,-72.640,-176.526,7.939,148.526
C05231=1183.265,320.844,-72.672,-176.523,7.942,148.527
C05232=1183.261,321.092,-72.703,-176.521,7.945,148.527
C05233=1183.257,321.340,-72.734,-176.519,7.949,148.527
C05234=1183.252,321.588,-72.766,-176.516,7.952,148.527
C05235=1183.248,321.836,-72.797,-176.514,7.955,148.527
C05236=1183.244,322.084,-72.828,-176.511,7.957,148.527
C05237=1183.240,322.332,-72.861,-176.509,7.960,148.527
C05238=1183.235,322.580,-72.892,-176.506,7.963,148.527
C05239=1183.231,322.828,-72.923,-176.504,7.966,148.527
C05240=1183.227,323.075,-72.955,-176.501,7.970,148.527
C05241=1183.223,323.324,-72.986,-176.499,7.973,148.527
C05242=1183.219,323.572,-73.018,-176.496,7.976,148.528
C05243=1183.215,323.819,-73.049,-176.494,7.979,148.528
C05244=1183.210,324.068,-73.081,-176.492,7.982,148.528
C05245=1183.206,324.316,-73.113,-176.489,7.985,148.528
C05246=1183.202,324.564,-73.144,-176.487,7.989,148.528
C05247=1183.198,324.812,-73.176,-176.484,7.992,148.528
C05248=1183.194,325.059,-73.208,-176.482,7.995,148.528
C05249=1183.189,325.308,-73.239,-176.479,7.998,148.528
C05250=1183.185,325.555,-73.271,-176.477,8.000,148.528
C05251=1183.181,325.804,-73.303,-176.474,8.003,148.528
C05252=1183.178,326.052,-73.335,-176.472,8.007,148.529
C05253=1183.173,326.299,-73.367,-176.469,8.010,148.529
C05254=1183.169,326.548,-73.398,-176.467,8.013,148.529
C05255=1183.164,326.795,-73.429,-176.465,8.016,148.529
C05256=1183.161,327.043,-73.461,-176.462,8.019,148.529
C05257=1183.156,327.292,-73.494,-176.460,8.023,148.529
C05258=1183.152,327.539,-73.525,-176.457,8.026,148.529
C05259=1183.148,327.787,-73.557,-176.455,8.029,148.529
C05260=1183.144,328.035,-73.589,-176.452,8.032,148.529
C05261=1183.139,328.283,-73.621,-176.450,8.035,148.530
C05262=1183.136,328.531,-73.653,-176.447,8.038,148.530
C05263=1183.132,328.779,-73.685,-176.445,8.042,148.530
C05264=1183.127,329.026,-73.717,-176.443,8.045,148.530
C05265=1183.123,329.274,-73.748,-176.440,8.048,148.530
C05266=1183.119,329.523,-73.781,-176.438,8.051,148.530
C05267=1183.114,329.770,-73.812,-176.436,8.053,148.530
C05268=1183.111,330.018,-73.844,-176.433,8.057,148.530
C05269=1183.106,330.266,-73.877,-176.431,8.060,148.531
C05270=1183.102,330.514,-73.908,-176.428,8.063,148.531
C05271=1183.098,330.762,-73.940,-176.426,8.066,148.531
C05272=1183.094,331.010,-73.972,-176.424,8.070,148.531
C05273=1183.090,331.258,-74.004,-176.421,8.073,148.531
C05274=1183.085,331.506,-74.036,-176.419,8.076,148.531
C05275=1183.082,331.753,-74.069,-176.416,8.079,148.531
C05276=1183.077,332.002,-74.101,-176.414,8.082,148.531
C05277=1183.073,332.249,-74.133,-176.412,8.086,148.532
C05278=1183.069,332.497,-74.165,-176.409,8.089,148.532
C05279=1183.065,332.745,-74.197,-176.407,8.092,148.532
C05280=1183.061,332.993,-74.229,-176.405,8.095,148.532
C05281=1183.056,333.240,-74.262,-176.402,8.098,148.532
C05282=1183.053,333.488,-74.294,-176.400,8.102,148.532
C05283=1183.048,333.737,-74.326,-176.397,8.105,148.532
C05284=1183.045,333.985,-74.358,-176.395,8.108,148.532
C05285=1183.040,334.233,-74.391,-176.392,8.111,148.533
C05286=1183.035,334.480,-74.423,-176.390,8.115,148.533
C05287=1183.032,334.728,-74.455,-176.388,8.118,148.533
C05288=1183.027,334.976,-74.488,-176.385,8.121,148.533
C05289=1183.024,335.224,-74.520,-176.383,8.124,148.533
C05290=1183.019,335.472,-74.552,-176.381,8.128,148.534
C05291=1183.015,335.719,-74.585,-176.378,8.130,148.533
C05292=1183.011,335.967,-74.617,-176.376,8.133,148.534
C05293=1183.007,336.216,-74.649,-176.374,8.136,148.534
C05294=1183.003,336.463,-74.682,-176.372,8.140,148.534
C05295=1182.999,336.712,-74.714,-176.369,8.143,148.534
C05296=1182.994,336.959,-74.746,-176.367,8.146,148.534
C05297=1182.990,337.207,-74.779,-176.364,8.149,148.535
C05298=1182.986,337.455,-74.811,-176.362,8.153,148.535
C05299=1182.982,337.702,-74.844,-176.359,8.156,148.535
C05300=1182.978,337.951,-74.877,-176.357,8.159,148.535
C05301=1182.974,338.198,-74.909,-176.355,8.162,148.535
C05302=1182.970,338.447,-74.942,-176.353,8.166,148.535
C05303=1182.965,338.694,-74.974,-176.350,8.169,148.536
C05304=1182.962,338.942,-75.006,-176.348,8.172,148.536
C05305=1182.957,339.189,-75.039,-176.345,8.175,148.536
C05306=1182.953,339.438,-75.072,-176.343,8.178,148.536
C05307=1182.950,339.685,-75.104,-176.341,8.182,148.536
C05308=1182.944,339.964,-75.141,-176.338,8.186,148.537
C05309=1182.940,340.243,-75.178,-176.335,8.189,148.537
C05310=1182.935,340.523,-75.215,-176.333,8.193,148.537
C05311=1182.931,340.801,-75.251,-176.330,8.196,148.537
C05312=1182.926,341.049,-75.285,-176.328,8.200,148.537
C05313=1182.923,341.297,-75.316,-176.326,8.203,148.537
C05314=1182.919,341.545,-75.350,-176.324,8.206,148.538
C05315=1182.914,341.792,-75.382,-176.321,8.210,148.538
C05316=1182.909,342.040,-75.415,-176.319,8.213,148.538
C05317=1182.905,342.288,-75.448,-176.316,8.216,148.538
C05318=1182.902,342.535,-75.481,-176.314,8.219,148.538
C05319=1182.898,342.783,-75.514,-176.312,8.223,148.539
C05320=1182.893,343.031,-75.546,-176.310,8.226,148.539
C05321=1182.889,343.279,-75.579,-176.307,8.229,148.539
C05322=1182.885,343.527,-75.612,-176.305,8.233,148.539
C05323=1182.881,343.775,-75.646,-176.303,8.236,148.539
C05324=1182.877,344.023,-75.677,-176.301,8.239,148.540
C05325=1182.873,344.270,-75.711,-176.298,8.243,148.540
C05326=1182.869,344.518,-75.744,-176.296,8.246,148.540
C05327=1182.865,344.766,-75.777,-176.294,8.249,148.540
C05328=1182.861,345.014,-75.810,-176.291,8.252,148.540
C05329=1182.856,345.262,-75.843,-176.289,8.256,148.541
C05330=1182.852,345.510,-75.876,-176.287,8.259,148.541
C05331=1182.848,345.757,-75.909,-176.285,8.262,148.541
C05332=1182.844,346.005,-75.941,-176.282,8.266,148.541
C05333=1182.840,346.253,-75.975,-176.280,8.269,148.542
C05334=1182.836,346.500,-76.008,-176.278,8.272,148.542
C05335=1182.832,346.748,-76.041,-176.276,8.276,148.542
C05336=1182.828,346.996,-76.074,-176.273,8.279,148.542
C05337=1182.824,347.243,-76.107,-176.271,8.282,148.542
C05338=1182.820,347.491,-76.140,-176.269,8.286,148.543
C05339=1182.816,347.739,-76.173,-176.267,8.289,148.543
C05340=1182.811,347.987,-76.207,-176.264,8.292,148.543
C05341=1182.807,348.234,-76.240,-176.262,8.296,148.543
C05342=1182.803,348.482,-76.273,-176.260,8.299,148.544
C05343=1182.799,348.730,-76.306,-176.258,8.302,148.544
C05344=1182.795,348.978,-76.339,-176.255,8.306,148.544
C05345=1182.791,349.225,-76.372,-176.253,8.309,148.544
C05346=1182.787,349.473,-76.406,-176.251,8.312,148.545
C05347=1182.783,349.721,-76.439,-176.249,8.316,148.545
C05348=1182.779,349.969,-76.472,-176.247,8.319,148.545
C05349=1182.775,350.217,-76.505,-176.244,8.322,148.545
C05350=1182.771,350.465,-76.539,-176.242,8.326,148.546
C05351=1182.766,350.712,-76.572,-176.240,8.329,148.546
C05352=1182.762,350.960,-76.605,-176.238,8.332,148.546
C05353=1182.758,351.207,-76.639,-176.236,8.336,148.546
C05354=1182.754,351.455,-76.673,-176.234,8.339,148.547
C05355=1182.749,351.703,-76.706,-176.231,8.343,148.547
C05356=1182.745,351.951,-76.739,-176.229,8.346,148.547
C05357=1182.742,352.199,-76.772,-176.227,8.349,148.547
C05358=1182.738,352.446,-76.806,-176.225,8.353,148.547
C05359=1182.734,352.694,-76.839,-176.223,8.356,148.548
C05360=1182.730,352.942,-76.873,-176.221,8.359,148.548
C05361=1182.726,353.189,-76.906,-176.218,8.363,148.548
C05362=1182.721,353.437,-76.940,-176.216,8.366,148.549
C05363=1182.717,353.685,-76.973,-176.214,8.370,148.549
C05364=1182.713,353.933,-77.007,-176.212,8.373,148.549
C05365=1182.709,354.181,-77.040,-176.210,8.376,148.549
C05366=1182.705,354.428,-77.074,-176.207,8.381,148.550
C05367=1182.701,354.676,-77.107,-176.205,8.384,148.550
C05368=1182.697,354.923,-77.141,-176.203,8.387,148.550
C05369=1182.693,355.171,-77.175,-176.201,8.391,148.551
C05370=1182.689,355.419,-77.208,-176.199,8.394,148.551
C05371=1182.685,355.666,-77.242,-176.196,8.398,148.551
C05372=1182.681,355.914,-77.275,-176.194,8.401,148.551
C05373=1182.676,356.162,-77.309,-176.192,8.405,148.552
C05374=1182.673,356.410,-77.343,-176.190,8.408,148.552
C05375=1182.669,356.658,-77.376,-176.188,8.412,148.553
C05376=1182.665,356.905,-77.410,-176.186,8.415,148.553
C05377=1182.660,357.153,-77.444,-176.184,8.418,148.553
C05378=1182.656,357.400,-77.478,-176.182,8.422,148.553
C05379=1182.653,357.648,-77.511,-176.180,8.425,148.554
C05380=1182.648,357.896,-77.546,-176.178,8.429,148.554
C05381=1182.644,358.143,-77.579,-176.176,8.432,148.554
C05382=1182.640,358.390,-77.613,-176.173,8.435,148.555
C05383=1182.637,358.639,-77.646,-176.172,8.439,148.555
C05384=1182.632,358.886,-77.681,-176.169,8.442,148.555
C05385=1182.628,359.134,-77.714,-176.167,8.446,148.556
C05386=1182.625,359.382,-77.748,-176.165,8.449,148.556
C05387=1182.620,359.629,-77.783,-176.163,8.453,148.556
C05388=1182.616,359.877,-77.816,-176.161,8.456,148.556
C05389=1182.611,360.124,-77.850,-176.159,8.460,148.557
C05390=1182.608,360.373,-77.884,-176.158,8.463,148.557
C05391=1182.604,360.620,-77.918,-176.155,8.467,148.558
C05392=1182.599,360.867,-77.952,-176.153,8.470,148.558
C05393=1182.596,361.116,-77.986,-176.151,8.474,148.558
C05394=1182.592,361.363,-78.020,-176.149,8.477,148.559
C05395=1182.588,361.610,-78.054,-176.148,8.481,148.559
C05396=1182.584,361.858,-78.088,-176.145,8.484,148.559
C05397=1182.579,362.106,-78.122,-176.143,8.488,148.560
C05398=1182.576,362.353,-78.156,-176.142,8.491,148.560
C05399=1182.572,362.601,-78.190,-176.139,8.495,148.560
C05400=1182.568,362.849,-78.225,-176.138,8.498,148.561
C05401=1182.564,363.096,-78.258,-176.136,8.502,148.561
C05402=1182.560,363.344,-78.293,-176.134,8.506,148.562
C05403=1182.556,363.592,-78.326,-176.132,8.509,148.562
C05404=1182.551,363.839,-78.361,-176.130,8.513,148.562
C05405=1182.548,364.087,-78.394,-176.128,8.516,148.563
C05406=1182.543,364.335,-78.429,-176.127,8.519,148.563
C05407=1182.539,364.582,-78.463,-176.125,8.523,148.564
C05408=1182.535,364.830,-78.498,-176.123,8.526,148.564
C05409=1182.532,365.077,-78.531,-176.121,8.530,148.564
C05410=1182.528,365.325,-78.566,-176.119,8.533,148.565
C05411=1182.524,365.572,-78.600,-176.117,8.537,148.565
C05412=1182.519,365.855,-78.639,-176.115,8.540,148.566
C05413=1182.514,366.136,-78.678,-176.114,8.545,148.566
C05414=1182.510,366.418,-78.717,-176.112,8.549,148.567
C05415=1182.505,366.699,-78.756,-176.110,8.552,148.567
C05416=1182.501,366.946,-78.791,-176.108,8.556,148.568
C05417=1182.498,367.194,-78.825,-176.106,8.560,148.568
C05418=1182.493,367.442,-78.859,-176.104,8.563,148.568
C05419=1182.489,367.689,-78.893,-176.103,8.567,148.569
C05420=1182.485,367.937,-78.928,-176.101,8.571,148.569
C05421=1182.481,368.184,-78.962,-176.100,8.573,148.570
C05422=1182.477,368.432,-78.997,-176.098,8.577,148.570
C05423=1182.473,368.679,-79.031,-176.096,8.581,148.571
C05424=1182.470,368.927,-79.065,-176.095,8.584,148.571
C05425=1182.465,369.175,-79.100,-176.093,8.587,148.572
C05426=1182.460,369.422,-79.134,-176.091,8.591,148.572
C05427=1182.457,369.670,-79.169,-176.090,8.595,148.572
C05428=1182.453,369.917,-79.203,-176.088,8.598,148.573
C05429=1182.449,370.165,-79.238,-176.087,8.601,148.573
C05430=1182.445,370.412,-79.272,-176.085,8.605,148.574
C05431=1182.441,370.660,-79.307,-176.083,8.608,148.574
C05432=1182.437,370.907,-79.342,-176.082,8.612,148.575
C05433=1182.433,371.155,-79.376,-176.081,8.615,148.575
C05434=1182.429,371.403,-79.410,-176.079,8.619,148.576
C05435=1182.425,371.651,-79.445,-176.077,8.622,148.576
C05436=1182.421,371.898,-79.479,-176.076,8.626,148.577
C05437=1182.417,372.145,-79.515,-176.074,8.629,148.577
C05438=1182.413,372.393,-79.549,-176.073,8.633,148.578
C05439=1182.409,372.641,-79.584,-176.072,8.636,148.578
C05440=1182.405,372.888,-79.618,-176.070,8.639,148.579
C05441=1182.401,373.136,-79.653,-176.069,8.643,148.579
C05442=1182.397,373.383,-79.688,-176.067,8.646,148.580
C05443=1182.393,373.631,-79.723,-176.066,8.650,148.580
C05444=1182.389,373.878,-79.757,-176.065,8.653,148.581
C05445=1182.385,374.126,-79.792,-176.063,8.657,148.581
C05446=1182.381,374.373,-79.827,-176.062,8.660,148.582
C05447=1182.377,374.621,-79.861,-176.061,8.664,148.582
C05448=1182.373,374.868,-79.895,-176.060,8.667,148.583
C05449=1182.369,375.116,-79.931,-176.058,8.670,148.583
C05450=1182.365,375.363,-79.965,-176.057,8.673,148.584
C05451=1182.361,375.611,-80.000,-176.055,8.677,148.584
C05452=1182.357,375.859,-80.036,-176.055,8.680,148.585
C05453=1182.353,376.106,-80.070,-176.053,8.684,148.586
C05454=1182.349,376.354,-80.104,-176.052,8.687,148.586
C05455=1182.345,376.601,-80.140,-176.051,8.691,148.587
C05456=1182.341,376.849,-80.174,-176.050,8.694,148.587
C05457=1182.337,377.096,-80.210,-176.048,8.697,148.588
C05458=1182.333,377.344,-80.244,-176.047,8.701,148.588
C05459=1182.329,377.592,-80.279,-176.046,8.704,148.589
C05460=1182.325,377.839,-80.314,-176.045,8.708,148.589
C05461=1182.321,378.087,-80.349,-176.044,8.710,148.590
C05462=1182.317,378.333,-80.384,-176.042,8.714,148.590
C05463=1182.313,378.582,-80.419,-176.042,8.717,148.591
C05464=1182.309,378.828,-80.454,-176.041,8.720,148.592
C05465=1182.305,379.077,-80.489,-176.039,8.724,148.592
C05466=1182.301,379.324,-80.524,-176.039,8.727,148.593
C05467=1182.297,379.571,-80.559,-176.037,8.730,148.593
C05468=1182.293,379.819,-80.594,-176.036,8.733,148.594
C05469=1182.288,380.066,-80.629,-176.035,8.737,148.594
C05470=1182.285,380.314,-80.664,-176.034,8.740,148.595
C05471=1182.282,380.562,-80.698,-176.033,8.743,148.596
C05472=1182.277,380.808,-80.734,-176.033,8.747,148.596
C05473=1182.273,381.057,-80.769,-176.031,8.750,148.597
C05474=1182.270,381.304,-80.804,-176.030,8.754,148.597
C05475=1182.265,381.552,-80.839,-176.030,8.757,148.598
